(* IEC 61131-3 sources: NachHouse_CORE/V200/APP (part 8) *)

(*
   If yes = false THEN
      yTx2 := '';
      _Nh1RowTxt();
   END_IF;
*)

END_FUNCTION
(*
FUNCTION _Nh_IO4 {HIDDEN} :BOOL
	// ACT,ALA,BLK - vykona sa pred SCN. SCN mozu vstupovat do ACT....
//   _Nh_IO_INI( vz:=4);
	FOR nd := 1 TO aVaz[cf].Rec DO
		IF _NhxVaz(cv:=4, nd:=nd) THEN
//			_Nh_IO_OK();

			ok := true;
  			IF _NhxPt(c:=xVaz^.in.c,n:=xVaz^.in.n,x:=22) THEN
			  	xDev  := xPt;
			ELSE
				ok := false;
			END_IF;
	      IF _NhxPt(c:=xVaz^.ou.c,n:=xVaz^.ou.n,x:=23) THEN
				xDev2 := xPt;
			ELSE
				ok := false;
			END_IF;
			IF ok THEN
		      xDev^.al.lst   := true;                                             				// SCN ma list
   	   	xDev2^.al.lst  := true;                                             				// DEV do scn ma list
      		IF xDev^.al.ou.cmd > 0 THEN
   	   	   xDev2^.al.IN.cmd  := xDev^.al.ou.cmd;
		         xDev2^.al.IN.par  := xVaz^.ou.p;                               				// do DEV sa posle vzdy parameter ou.p
//	         xDev2^.al.IN.par  := 8;                               				// do DEV sa posle vzdy parameter ou.p

   	   	   xDev2^.al.IN.val  := xDev^.al.ou.val;                       					// parameter DEV z vazby
      		   xDev2^.al.wsb  	:= xDev^.al.wsb;                       						// zaisi pripadne blokovanie PIR pte DEV v liste
					xDev^.al.wsb		:= false;																// po prebrati vynuluje priznak WSB
		      END_IF;
			END_IF;
		END_IF;
   END_FOR;
END_FUNCTION
*)

FUNCTION _Nh_IO4  {HIDDEN}  :BOOL
	// ACT,ALA,BLK - vykona sa pred SCN. SCN mozu vstupovat do ACT....
   _Nh_IO_INI( vz:=4);
	FOR nd := 1 TO aVaz[cf].Rec DO
		IF _Nh_IO_OK() THEN
	      xDev^.al.lst   := true;                                             				// SCN ma list
      	xDev2^.al.lst  := true;                                             				// DEV do scn ma list
      	IF xDev^.al.ou.cmd > 0 THEN
   	      xDev2^.al.IN.cmd  := xDev^.al.ou.cmd;
	         xDev2^.al.IN.par  := xVaz^.ou.p;                               				// do DEV sa posle vzdy parameter ou.p
      	   xDev2^.al.IN.val  := xDev^.al.ou.val;                       					// parameter DEV z vazby
      	   xDev2^.al.wsb  	:= xDev^.al.wsb;                       						// zaisi pripadne blokovanie PIR pte DEV v liste
				// toto sa urovni az akcii v dalsom cykle
//				xDev^.al.wsb		:= false;																// po prebrati vynuluje priznak WSB
	      END_IF;
		END_IF;
   END_FOR;
END_FUNCTION

// z akcii uz vypinaju aj scenu ak je lvl=0.0 alebo ak < 100, tak zapnu len tie DEV pomerom, ktore maju v par, lvl > 0.0
FUNCTION _Nh_IO3    :BOOL
	// SCN - po ACT,(IO4) ktore mozu nastavit SCN nejaky stav
   _Nh_IO_INI( vz:=3);
	FOR nd := 1 TO aVaz[cf].Rec DO
		IF _Nh_IO_OK() THEN
	      xDev^.al.lst   := true;                                             					// SCN ma list
      	xDev2^.al.lst  := true;                                             					// DEV do scn ma list
			xScn				:= xDev;
      	IF xDev^.al.ou.cmd > 0 THEN
				IF xDev^.cf.typ = 1 THEN
      		   xDev2^.al.up  		:= xDev^.al.up;                       						// parameter DEV z vazby
					xDev2^.al.IN.cmd  := xDev^.al.ou.cmd;
		         xDev2^.al.IN.par  := xVaz^.ou.p;                               					// do DEV sa posle vzdy parameter ou.p
				ELSE
		         xDev2^.al.IN.par  := xVaz^.ou.p;                               					// do DEV sa posle vzdy parameter ou.p
   	   	   xDev2^.al.IN.val  := xDev^.al.ou.val;                       						// parameter DEV z vazby
					xDev2^.al.IN.cmd  := xDev^.al.ou.cmd;
(*
				IF xDev^.al.ou.val = 0.0 THEN
	   	      xDev2^.al.IN.cmd  := 10;
				ELSIF xDev^.al.ou.val < 100.0 THEN
	   	      xDev2^.al.IN.cmd  := 9;
					xDev^.al.Qx 		:= false;
				ELSE
	   	      xDev2^.al.IN.cmd  := xDev^.al.ou.cmd;
				END_IF;
      	   xDev2^.al.wsb  	:= xDev^.al.Wsb;                       						// parameter DEV z vazby
*)

					IF xDev^.al.ou.cmd = 11 THEN
						IF aCfg[xVaz^.ou.c].par > 0 THEN															// DEV v scene ma parameter
							IF _NhxPar(cp := aCfg[xVaz^.ou.c].par, np := xVaz^.ou.p,x:=252) = false  THEN																	   // NEnasiel sa parameter
							;
							ELSIF xPar^.all.lvl = 0 THEN						// LVL>0 ale ine ako ma byt
	   	      			xDev2^.al.IN.cmd  := 10;
							END_IF;
						END_IF;
					END_IF;
      		   xDev2^.al.wsb  	:= xDev^.al.Wsb;                       						// parameter DEV z vazby
				END_IF;
			ELSIF xDev^.cf.typ = 1 THEN																	// len rolety
				IF xDev2^.al.sta > 2  THEN
					xScn^.cx.all.LastScnOn := true;
				END_IF;
			ELSIF xDev2^.al.ou.val > 0. THEN
				xScn^.cx.all.LastScnOn := true;
(*
			ELSIF xDev^.al.Qx = false THEN																// DEV v scene je zapnute
				;
			ELSIF aCfg[xVaz^.ou.c].par > 0 THEN															// DEV v scene ma parameter
				IF _NhxPar(cp := aCfg[xVaz^.ou.c].par, np := xVaz^.ou.p,x:=252) = false  THEN																	   // NEnasiel sa parameter
					;
				ELSIF xPar^.all.lvl <> REAL_TO_USINT(xDev2^.al.ou.val) THEN						// LVL>0 ale ine ako ma byt
					// vypne scenu
//					xDev^.al.In.val 	:= 0.0;	//xDev2^.al.ou.val;
//					xDev^.al.Ou.val 	:= 0.0;	//xDev2^.al.ou.val;
					xDev^.al.Qx 		:= false;
					xDev^.al.in.cmd	:= 3;																	// vypne priznak zapnutia a resetne casy
				END_IF;
*)
			END_IF;
		END_IF;
   END_FOR;
END_FUNCTION

(*
// z akcii uz vypinaju aj scenu ak je lvl=0.0 alebo ak < 100, tak zapnu len tie DEV pomerom, ktore maju v par, lvl > 0.0
FUNCTION _Nh_IO3    :BOOL
	// SCN - po ACT,(IO4) ktore mozu nastavit SCN nejaky stav
   _Nh_IO_INI( vz:=3);
	FOR nd := 1 TO aVaz[cf].Rec DO
		IF _Nh_IO_OK() THEN
	      xDev^.al.lst   := true;                                             					// SCN ma list
      	xDev2^.al.lst  := true;                                             					// DEV do scn ma list
			xScn				:= xDev;
      	IF xDev^.al.ou.cmd > 0 THEN
				IF aCfg[xVaz^.ou.c].par > 0 THEN															// DEV v scene ma parameter
					IF _NhxPar(cp := aCfg[xVaz^.ou.c].par, np := xVaz^.ou.p,x:=252) THEN
						xScn^.me.delayOff := MAX(xScn^.me.delayOff, _Nh_N12(aCfg[xVaz^.ou.c].tgrp=31,xPar^.all.tDelay,xPar^.all.tDelay/10)+2 );	// MAX opozdene spustenie z niektoreho DEV
					ELSE
						yTx2	:= CONCAT('_Nh_IO3: Not Find par: cf:',USINT_TO_STRING(xVaz^.ou.c),',cp:',USINT_TO_STRING(aCfg[xVaz^.ou.c].par),
											', np: ',INT_TO_STRING(xVaz^.ou.p),', vz3:',INT_TO_STRING(nd)  )  ;
    					rb		:= _Nh1RowTxt(logRst := 1);
						ok1 	:= false;
					END_IF;
				ELSE	ok1 := false;
				END_IF;
 				xDev2^.al.wsb  	:= xDev^.al.Wsb;                       						// priznak WSB
				xDev2^.al.IN.cmd  := xDev^.al.ou.cmd;
  	   	   xDev2^.al.IN.val  := xDev^.al.ou.val;                       					// parameter DEV z vazby
	         xDev2^.al.IN.par  := xVaz^.ou.p;
				IF xDev^.cf.typ = 1 THEN
      		   xDev2^.al.up  		:= xDev^.al.up;                      						// pre ROL DOLEZITE !!! - nastavi smer pohybu rolety
				END_IF;
				IF xDev^.al.ou.cmd = 11 THEN
					IF ok1 = false THEN
						;
					ELSIF xPar^.all.lvl = 0 THEN						// LVL>0 ale ine ako ma byt
 						xDev2^.al.IN.cmd  := 10;
					END_IF;
				END_IF;
			ELSIF xDev^.al.ou.val = 0. THEN																// scn je vypnuta
				;
			ELSIF xDev^.cf.typ = 1 THEN																	// len rolety
				IF xDev2^.al.sta > 2  THEN
					xScn^.cx.all.LastLvl	:= 100;
				END_IF;
			ELSIF xDev2^.al.ou.val > 0. THEN
				xScn^.cx.all.LastLvl	:= 100;
			END_IF;
		END_IF;
   END_FOR;
END_FUNCTION
*)

(*

// pred Rosochom - z akcii nevypinali scenu, ked bola 0.0

FUNCTION _Nh_IO3  :BOOL
	// SCN - po ACT,(IO4) ktore mozu nastavit SCN nejaky stav
   _Nh_IO_INI( vz:=3);
	FOR nd := 1 TO aVaz[cf].Rec DO
		IF _Nh_IO_OK() THEN
	      xDev^.al.lst   := true;                                             					// SCN ma list
      	xDev2^.al.lst  := true;                                             					// DEV do scn ma list
			xScn				:= xDev;
      	IF xDev^.al.ou.cmd > 0 THEN
	         xDev2^.al.IN.par  := xVaz^.ou.p;                               					// do DEV sa posle vzdy parameter ou.p
      	   xDev2^.al.IN.val  := xDev^.al.ou.val;                       						// parameter DEV z vazby
   	      xDev2^.al.IN.cmd  := xDev^.al.ou.cmd;
      	   xDev2^.al.wsb  	:= xDev^.al.Wsb;                       						// parameter DEV z vazby
			ELSIF xDev^.al.Qx = false THEN																// DEV v scene je zapnute
				;
			ELSIF aCfg[xVaz^.ou.c].par > 0 THEN															// DEV v scene ma parameter
				IF _NhxPar(cp := aCfg[xVaz^.ou.c].par, np := xVaz^.ou.p,x:=252) = false  THEN																	   // NEnasiel sa parameter
					;
				ELSIF xPar^.all.lvl <> REAL_TO_USINT(xDev2^.al.ou.val) THEN						// LVL>0 ale ine ako ma byt
					// vypne scenu
//					xDev^.al.In.val 	:= 0.0;	//xDev2^.al.ou.val;
//					xDev^.al.Ou.val 	:= 0.0;	//xDev2^.al.ou.val;
					xDev^.al.Qx 		:= false;
					xDev^.al.in.cmd	:= 3;																	// vypne priznak zapnutia a resetne casy
				END_IF;
			END_IF;
		END_IF;
   END_FOR;
END_FUNCTION
*)

(*
FUNCTION _Nh_IO3  :BOOL
	// SCN - po ACT,(IO4) ktore mozu nastavit SCN nejaky stav
   _Nh_IO_INI( vz:=3);
	FOR nd := 1 TO aVaz[cf].Rec DO
		IF _Nh_IO_OK() THEN
	      xDev^.al.lst   := true;                                             					// SCN ma list
      	xDev2^.al.lst  := true;                                             					// DEV do scn ma list
      	IF xDev^.al.ou.cmd > 0 THEN
   	      xDev2^.al.IN.cmd  := xDev^.al.ou.cmd;
	         xDev2^.al.IN.par  := xVaz^.ou.p;                               					// do DEV sa posle vzdy parameter ou.p
      	   xDev2^.al.IN.val  := xDev^.al.ou.val;                       						// parameter DEV z vazby
//      	   xDev2^.al.wsb  	:= xDev^.cx.all.LastWsb;                       						// parameter DEV z vazby
      	   xDev2^.al.wsb  	:= xDev^.al.Wsb;                       						// parameter DEV z vazby

//  	   	ELSIF xDev^.al.Qx THEN 												      						// test SCN ci je ON/OFF, povoli sa ked je scena v pokoji Qx=true
  	   	ELSIF xDev^.cx.all.LastScnOn THEN 												      						// test SCN ci je ON/OFF, povoli sa ked je scena v pokoji Qx=true
				// ak aspon jedno DEV nema hodotu aku ma mat v scene = vypne scenu
				IF xDev^.al.ou.val > 0.0  THEN																// scena je zapnuta
					IF aCfg[xVaz^.ou.c].par > 0 THEN															// DEV v scene ma parameter
    					IF _NhxPar(cp := aCfg[xVaz^.ou.c].par, np := xVaz^.ou.p,x:=252) = false THEN
							;
						ELSIF xPar^.all.lvl <> REAL_TO_USINT(xDev2^.al.ou.val) THEN						// kazde DEV v SCN-liste musi mat aktualny LVL = parametru

							xDev^.cx.all.LastScnOn	:= false;														// ak sa najde prva nezhoda, tato SCN sa oznaci a OFF
							xDev^.al.sta 				:= 0;                                              // a uz sa s nou tu nepracuje
							xDev^.al.IN.val 			:= 0.0;															// vypne scenu
							xDev^.al.OU.val 			:= 0.0;
      					/////15.9.24	vypne prebiehajuce casy vypnutia
//							xDev^.al.et 	:= 0;																	// cas od PIR
//							xDev^.al.ex 	:= 0;																	// max.cas zapnutia
						END_IF;
					END_IF;
				END_IF;
			END_IF;
		END_IF;
   END_FOR;
END_FUNCTION
*)

FUNCTION _Nh_SVX_CMD_1     : BOOL
	IF xDev^.al.in.CMD = 3 THEN         										// len nastavilo proznak vypnutia a resetlo casy
		;
	ELSIF xDev^.al.in.CMD > 0 THEN         										// povolene prikazy testuju blokovanie PIR a oneskorenie
			xDev^.al.Off 			:= xDev^.al.OU.val = 0.0 AND xDev^.al.IN.val > 0.0; // je vypnute a ma sa zapnut - pre lampu, ktora ma dlhy nabeh z OFF->ON
			xDev^.cx.all.LastWsb	:= xDev^.al.wsb;										// prisiel z wsb
			IF xDev^.al.RUN = 255 THEN   													// Koniec Delay
				xDev^.al.RUN := 0;
 			ELSIF xPar^.all.tDelay > 0 THEN 												// opozdene vykonanie
	   	   xDev^.al.RUN   	:= xDev^.al.in.CMD;                              			// po skonceni opozdenia sa zoberie LVL z parametri - tu pridu len DEV s parametrom
				xDev^.al.in.CMD	:= 0;
   	   	xDev^.al.et    	:= xPar^.all.tDelay ;                        //
  	   		xDev^.al.CM    	:= 2;                                        // vykonava sa opozdenie
   	   	xDev^.al.ct    	:= 3;                                     	// Delay je vzdy v [100ms]
   		END_IF;
		   IF xDev^.al.in.CMD = 1 THEN                                    	// prepnut WEB/WSB
         	xDev^.al.in.val   := vr;
      		IF xDev^.al.ou.val > 0.0 THEN                               	// je zapnute, treba vypnut z WEB/WSB
         		xDev^.al.in.val   := 0.0;
				ELSIF xPar^.all.lvl = 0 THEN
           		xDev^.al.in.val	:= 100.0;                              // zapnut naplno
					xPar^.all.lvl 		:= REAL_TO_USINT(xDev^.al.in.val);				// nastavi LVL v prametri - najma pri vazbach
      		ELSE
					xDev^.al.in.val := USINT_TO_REAL(xPar^.all.lvl);				// nastavi LVL v prametri - najma pri vazbach
      		END_IF;
      		_Nh_Dev_RMP();
   		END_IF;
		   IF xDev^.al.in.CMD > 0 THEN         										// povolene prikazy testuju blokovanie PIR a oneskorenie
			   _NhxRom(nr := xDev^.cf.rom, x:=-10);
			   IF xDev^.al.wsb = false THEN                                   // nic sa nedeje neprislo z WSB {mozno z ACT..SCN}
   			   ;
	   		ELSIF  xDev^.al.in.val > 0.0 AND xPar^.all.BlPirON THEN       	// je ON
   	   		xRom^.me.BlPirOn    := 50;  	                             	// zapnutie od WSB/WEB vzdy blokuje PIR
   	   		xRom^.me.BlPirOff   := 0;                               		// resetne sa cas blokovania po vypnuti
	   		ELSIF xPar^.all.BlPirOff AND xRom^.cx.BlPirOFF > 0 THEN 			// kontrola na blokovanie PIR po vypnuti WSB/WEB
   				xRom^.me.BlPirOff := MAX(xRom^.me.BlPirOff,xRom^.cx.BlPirOFF); // max cas blokovania po vypnuti
	   		END_IF;
				// casy vypnutia
	         IF xDev^.al.IN.val < 1.0 THEN                   		// ma sa vypnut
					xDev^.al.IN.val 	:= 0.0;
   	      ELSIF xDev^.al.OU.val < 1.0 THEN                      // je OFF a ma za zapnut
      	      xDev^.al.ex := UINT_TO_INT(xDev^.cx.all.tMaxON);   // max cas zapnutia [min] - pohyb neresetuje
         	END_IF;
	         IF xDev^.al.IN.val > 0.0 THEN
					xDev^.al.up		:= true;
      	      IF xPar^.all.tOff > 0 THEN
         	      xDev^.al.et := xPar^.all.tOff;                  // vypnut po cas
            	   xDev^.al.ct := 3;                               // po 100mSEC
	            ELSE
   	            xDev^.al.et := 0;                               // nema sa vypnut po case
      	      END_IF;
				ELSE
					xDev^.al.ex    	:= 0;
				 	xDev^.al.et    	:= 0;
				END_IF;
				_Nh_Dev_CMD();			                                 // vyvolat zapnutie HW cez CMD
			END_IF;
	END_IF;

END_FUNCTION

FUNCTION _Nh_SVX_Qx    : BOOL
	_Nh_SVX_Qx := false;
	IF _Dev_Qx_PAR(dpa:=xDev^.cf.par) THEN

		_Nh_SVX_Qx := true;
		xDev^.al.el		:=	0;
		xDev^.al.CM    := 0;													// ak bezi delay cm:=2, novy prikaz ho zrusi
//		xDev^.al.RUN   := 0;	                                    //

		IF aCfg[cf].par > 0 THEN											// dev ma parameter, SIR napr nema parameter
 	   	vr    := USINT_TO_REAL(xPar^.all.Lvl);                // default sa podhodi LVL
		ELSE
			vr := 0.0;                                          	// bez parametra nebude potrebovat, lebo pride konkretne CMD
		END_IF;

		xDev^.cx.all.LastCMD 	:= xDev^.al.in.CMD;					// zapamata posledny pokyn
// 		xDev^.cx.all.LastCMDin	:= true;                         // pokyn je prichadzajuci

		CASE xDev^.al.in.CMD OF
	      1: // prepnut z WEB
   	      xDev^.al.wsb      := true;									// nasilne sa podhodi ako z WSB, aby sa zablokoval pir
//      	   xDev^.al.in.CMD   := 1;
	      2: // prepnut z WSB												// wsb nastavi priznak WSB vo vazbach automaticky
   	      xDev^.al.in.CMD   := 1;
      	3: // resetovat casy nastavit OFF, ale neposielat nic
				cmd	:= 0;
				_Nh_Dev_OFF(cmd:=3);
				xDev^.al.in.CMD := 0;

			6: // stmievanie z  WSB - start
   	      IF xDev^.al.ou.VAL > 0.0 THEN								// stmieva sa len, ak je ON
      	      xDev^.al.Up    := NOT xDev^.al.Up;
					IF xDev^.al.ou.VAL <= 1.0 THEN
      	      	xDev^.al.Up    := true;
					ELSIF xDev^.al.ou.VAL > 99.0 THEN
    					xDev^.al.Up    := false;
					END_IF;
					IF aCfg[cf].lvl254 THEN
	         	   xDev^.al.rmp   := 1;                            // doladit ???
					ELSE
	         	   xDev^.al.rmp   := 3;
   				END_IF;
	  			ELSIF _NhxRom(nr := xDev^.cf.rom, x:=-13) THEN					// ak svetlo nesvieti, PRESS zrusi blokovanie
      	      xRom^.me.BlPirOn 	:= 0;
         	   xRom^.me.BlPirOff := 0;
					xDev^.al.cm := 255;								// aby sa uz az do pustenia BTN nic nerobilo
	         END_IF;
				xDev^.cx.all.LastLvl	:= REAL_TO_USINT(xDev^.al.Ou.val);
				xDev^.al.in.CMD		:= 0;

   	   7: // slider SVA
				IF aCfg[cf].lvl254 THEN
         	   xDev^.al.rmp   := 1;                            // doladit ???
				ELSE
         	   xDev^.al.rmp   := 2;
  				END_IF;
				xDev^.cx.all.LastLvl	:= REAL_TO_USINT(xDev^.al.Ou.val);
				xDev^.al.in.CMD		:= 0;
				xDev^.al.CM				:= 7;

	      8: // RGB - vyber farby a slidery RGBWA
   	      xDev^.al.rmp      := 0;
				xDev^.al.in.CMD	:= 0;

	      9: // specialne zapnutie/vypnutie
				// ak  je prichadzajuci LVL = 0, tak vypne,
				// ak lvl < 100 tak zapne na pomer k hodnoty z parametra
				// ak lvl = 100% tak zapne na plny parameter
				IF vr  = 0.0 THEN
					xDev^.al.in.val := 0.0;
				ELSIF xDev^.al.in.val < 100.0 THEN
					xDev^.al.in.val := vr * xDev^.al.in.val * 0.01;
				ELSE
					xDev^.al.in.val := vr;
				END_IF;
				_Nh_Dev_RMP();

	     10: // OFF + zapnut blokovanie PIR
   	      xDev^.al.in.val   := 0.0;

	     11: // zapnutie na 100%
				xDev^.al.in.val   := 100.0;                              // zapnut naplno
				_Nh_Dev_RMP();

	     12: // blikac - priame zapnutie na LVL z parametra ak al.in.val > 0, iba vypnut , bez kontroly casov
   	     	xDev^.al.IN.val   := vr;
      	   xDev^.al.wsb      := false;								// nasilne sa podhodi ako z WSB, aby sa zablokoval pir
				_Nh_Dev_RMP();

	     13: // zapnutie na to co je al.in.val (blikac), bez kontroly casov
				_Nh_Dev_RMP();

		  14: // zapnut na LVL, ulozenu v parametri, nastavit casy opozdeny start/po case vypnut/max.cas zapnutia
   	      xDev^.al.in.val   	:= vr;
				_Nh_Dev_RMP();

	     15: // len zapamatat/ulozit aktualnu LVL pre dalsiu obnovu (blikac)
				xDev^.cx.all.LastLvl := REAL_TO_USINT(xDev^.al.OU.Val);
				xDev^.al.in.CMD	:= 0;
				xDev^.al.trg.Q  	:= 0;													// aby CMD v dalom cykle vyhodnotilo ako Qr, nieQ
				xDev^.al.trg.Qf 	:= 0;

   	  16: // obnovit zapamatany LVL po ukonceni blikaca
				xDev^.al.In.Val		:= USINT_TO_REAL(xDev^.cx.all.LastLvl);
				_Nh_Dev_CMD();			                                 // vyvolat zapnutie HW cez CMD
				xDev^.al.in.CMD	:= 0;

	     21: // PIR - ON
   	      _NhxRom(nr := xDev^.cf.rom, x:=-14);
      	   IF xRom^.me.BlPirOn = 0 AND xRom^.me.BlPirOFF = 0 THEN  	// nie je blokovana ROM po vypnuti, ani po zapnuti
         	   IF xDev^.al.ou.Val < 0.9 OR xPar^.all.rPir THEN          	// je OFF alebo bezi cas-to-OFF a pohyb resetuje cas
            	   xDev^.al.IN.val   := vr;
						_Nh_Dev_RMP();
						xDev^.al.CM				:= 14;
   	         END_IF;
      	   ELSE
	      	   xDev^.al.in.CMD   := 0;
   	      END_IF;
      	   xDev^.al.wsb      := 0;

			{$IFDEF __NH_DALI}

   	   43: // ON/OFF DLS + dali 5 in On
				xDLs	:= xDev;
	         IF xDls^.cx.cfg.out5inOne THEN 										// 5 in On
					IF xDev^.al.OU.val > 0.0 THEN										// je zapnute, treba vypnut
						ii						:= 0;
					ELSE
						ii						:= 254;
					END_IF;
					FOR i := 1 TO 5 DO
						xPar^.rgb.lvl[i] := ii;          							// default parameter je namapovany
   	  			END_FOR;
					xDev^.al.in.val 	:= 100;                                // vzdy posle prikaz do DLM
	      	   xDev^.al.rmp      := 0;
					cmd					:= 143;
					xDev^.al.in.CMD	:= 0;
   	      ELSE

      	   END_IF;

	     143: // DLS 5-In-One pokyn z {TVE} nastavenych na RGBWA
				xPtIO 	:= UDINT_TO_PTR( REAL_TO_UDINT(xDev^.al.in.val) ) ;	   		// prenasa sa adresa IO, pre zistenie farby
				IF xPtIO^.val > 0. THEN																	// zapnut
					ii	:= 254;
				ELSE
					ii	:= 0;
				END_IF;
				IF xPtIO^.dev.o > 0 THEN                                                // zisti sa, ktora farba sa nastavika
//						xPar^.rgb.lvl[xPtIO^.dev.o] := MIN(254,REAL_TO_USINT(xPtIO^.val));   // nastavi sa LVL, vzdy 254
					xPar^.rgb.lvl[xPtIO^.dev.o] := ii;   											// nastavi sa LVL, konkretnehj farby RGBWA vzdy 254
				END_IF;
//				xDev^.al.in.val	:= 255.0;                                               // vzdy vysle sa prikaz - aktualizuje vsetky farby
				xDev^.al.in.val 	:= 100;                                // vzdy posle prikaz do DLM
				cmd					:= 143;
				xDev^.al.in.CMD	:= 0;

	     144: // DLS 5-In-One dotyk nad konkretnou farbou znamen vyslat to co tam je
//				xDev^.al.in.val 	:= 255.0;
				xDev^.al.in.val 	:= 100;                                // vzdy posle prikaz do DLM
				xDev^.al.in.CMD	:= 0;
   	   	cmd       			:= 143;
			{$END_IF}
   	ELSE
			;
   	END_CASE;
//		_Nh_SVX_CMD_1();

	ELSIF xDev^.al.trg.Q THEN                                         // presss alebo len zopar cyklov, ked sa neuvolni cmd

		IF aCfg[cf].lvl254 THEN	                                       // DALI
			ok	 	:= (SYSTEM_S.R_EDGE_500MS OR SYSTEM_S.F_EDGE_500MS);  // vysiela sa kazdy 250ms
			kr 	:= 7.;
//			kr 	:= 1.;
			ur		:= 100.;
		ELSE
			ok	 	:= aSys.PULSE_50MS;	//SYSTEM_S.R_EDGE_100MS;			// kazdych 50ms, alebo podla cyklu
			kr 	:= 1.;
			ur		:= 100.;
		END_IF;

		IF xDev^.al.up = false THEN
			kr	:= kr * -1.;
		END_IF;
		cmd	:= 0;
		IF xDev^.al.cm = 255 THEN                                      // press, ked svetlo nesvietilo {zrusenie blokovania}
			;
		ELSIF ok = false THEN														// nenastala casova vzorka
			;
		ELSIF xDev^.cx.all.LastCMD = 6 THEN										// drzi sa WSB
			vr						:= xDev^.al.IN.val + kr ;
  			IF vr > 100. THEN
				vr := 100.;
			ELSIF vr < 1. THEN
				vr := 1.;
			END_IF;
			xDev^.al.IN.val	:= LIMIT(1.0, vr, ur);
			IF vr <> xDev^.al.IN.val THEN                              	// uz sa dosiahol niektory limit
				xDev^.al.cm := 255;
			ELSE
				_Nh_Dev_CMD();
			END_IF;
		ELSIF xDev^.cx.all.LastCMD = 7 THEN	                           // slider
			IF ABS(xDev^.al.ou.val - xDev^.al.In.val) >= ABS(kr)  THEN  // bude vysielat do HW, len ked je zmena vacsia
	 			_Nh_Dev_CMD();
			END_IF;
		ELSIF xDev^.cx.all.LastCMD = 8 THEN	                           // RGB
 			_Nh_Dev_CMD();
		END_IF;

	ELSIF xDev^.al.trg.Qf THEN														// koniec CMD
		xDev^.al.wsb 	:= 0;
		IF xDev^.cx.all.LastCMD = 8 	OR									// zmena fazby = vyber predvolby
			xDev^.al.cm = 255				OR                         // prikaz uz bol vykonany
			(xDev^.cx.all.LastCMD >= 4 AND xDev^.cx.all.LastCMD <= 7) THEN	// 4=SW-Dim,6=WSB-dim,7-slider
			xDev^.al.cm		:= 0;
			xDev^.al.et		:= 0;

//			_NhxPar(cp := aCfg[cf].par , np := xDev^.al.ou.par, cf:=cf, nd:=nd, x:=110);

			xPar^.all.lvl := REAL_TO_USINT(xDev^.al.in.val);		// zapamata LVL v default parametri
			_Nh_Dev_CMD();														// este raz posle, lebo slider nemusel zachytit vsetko
		END_IF;

	ELSIF aSys.Restart THEN
		IF xDev^.cf.LvlOnRst  THEN	 								// po restarte obnovit
			_Nh_Dev_CMD();			                                 // zapnut HW
		ELSE
//			xDev^.al.in.Val := 0.0;                               // vypnut aj IN
		END_IF;
	END_IF;
END_FUNCTION

FUNCTION _Nh_SVX   : BOOL
	VAR_INPUT
		c		: 	USINT;
	END_VAR
	VAR_TEMP
		i		: USINT;
//		ii		: USINT;
	END_VAR
   _Nh_SVX	:= _Dev_INI(c := c);
	nd			:= 1;
   WHILE nd <= aCfg[cf].Rec DO
      IF _Nh_Dev_REC(blk:=true) THEN //AND nd = 2 THEN
			IF _Nh_SVX_Qx() THEN
				_Nh_SVX_CMD_1();																// nie pre SCN
			END_IF;
		   xDev^.al.IN.CMD   := 0;															// reset vstup, aby s v dalsom kole vyhodnotil Q,Qf
			IF xDev^.al.cm = 2 THEN
				cmd	:= 0;
				IF _Nh_Dev_ET_UINT(t :=3, et:= ADR(xDev^.al.et) ) THEN			// odpocitava Delay [min]
					xDev^.al.in.cmd	:= xDev^.cx.all.LastCMD;
					xDev^.al.in.par	:= xDev^.al.ou.par;
					xDev^.al.RUN		:= 255;
//					xDev^.al.cm 		:= 0;
				END_IF;
			ELSIF xDev^.al.cm = 255 THEN													// bezi press a uz sa nema co vykonat
				cmd	:= 0;
			ELSIF _Nh_Dev_ET_UINT(t :=3, et:= ADR(xDev^.al.et) ) OR				// odpocitava cas zapnutia [min]
 					_Nh_Dev_ET_INT (t :=2, et:= ADR(xDev^.al.ex) ) THEN			// odpocitava max cas zapnutia [min]
				_Nh_Dev_OFF(cmd:=0);
				_Nh_Dev_CMD();			                                 			// zapnut HW
			END_IF;
//			ok3	:= true;
			ok3	:= cf <> 42;																// stav DALI-mastra sa robi inak ako cez _Nh_Sta_Rom
			CASE cmd OF
           	 0: ;
				 3: ; //
          	10: ; // SVD,ZAS,SIR.... digital
			      	xSvD 					:= xDev;
						IF xSvD^.hw.d[0] > 0 THEN
	                  xDev^.al.Ou.CMD	:= 180;
   	   			   xPtB 					:= UDINT_TO_PTR(xSvD^.hw.d[0]);

 							_Nh_Log_Evn_ADD(tsk:=10);

      				   xDev^.al.OU.val   := xDev^.al.IN.val;
         			 	xPtB^             := REAL_TO_BOOL(xDev^.al.OU.val);                  // in, nie ou
	 	      		   IF xDev^.cf.inv THEN
 		         			xPtB^ := NOT xPtB^;
	      	  	   	END_IF;
						END_IF;

				11:	// SVA
    					xDev^.al.Ou.CMD	:= 180; 																	// default CMD pre vystupne zariadenie
						IF xDev^.hw.typ = 43 THEN
							;
						ELSIF xDev^.hw.d[0] > 0  THEN                                     			// xDev = xSva
							ok := xDev^.cx.dim.DimHW;
							IF ok THEN                                                        // ma sa stmievat HW
								IF xDev^.hw.d[1] = 0 THEN                                     	// ak nie je HW adresa stmievania
									ok := false;                                                // bude sa stmievat SW
								END_IF;
							ELSIF xDev^.hw.d[1] > 0 THEN                                     	// ma sa stmievat SW ale mame HW adresu rampy
								xPtU 					:= UDINT_TO_PTR(xDev^.hw.d[1]);
								xPtU^ 				:= 0;														// rampu nastavi na 0
							END_IF;

 							_Nh_Log_Evn_ADD(tsk:=10);

							IF ok THEN
								xPtU 					:= UDINT_TO_PTR(xDev^.hw.d[1]);
								xPtU^ 				:= xDev^.al.rmp;
   	   		         xDev^.al.ou.val   := xDev^.al.in.val;
							ELSE
								_Nh_Dim_SW();
							END_IF;
							xDev^.al.el			:= 0;
							xPtR 					:= UDINT_TO_PTR(xDev^.hw.d[0]);
							xDev^.al.ou.val	:= LIMIT(0.0, xDev^.al.in.val, 100.0);
							xPtR^					:= _Nh_LVL_100(	lvlMin	:=	xDev^.cx.sva.Lv0,
																			lvlMax	:=	xDev^.cx.sva.Lv1,
																			lvlIn		:=	xDev^.al.ou.val);
							CASE xDev^.hw.typ OF
      	              0:	// BOOL
									xPtB	:= xPtr;
									xPtB^	:= REAL_TO_BOOL(xPtr^);
                    	  1: // REAL
//							  		xPtR^	:= kr;
							  2:	// USINT
									xPtU	:= xPtr;
									xPtU^	:= REAL_TO_USINT(xPtr^);
      	            END_CASE;
						END_IF;

(*

                  xDev^.al.Ou.CMD	:= 180; 																	// default CMD pre vystupne zariadenie
						IF xDev^.hw.d[2] > 0 THEN                                     		// mame adresu HW minima (RLC)
 							xPtR 	:= UDINT_TO_PTR(xDev^.hw.d[2]);
							xPtR^ := _Nh_255_100(xDev^.cx.sva.Lv0);
						END_IF;
						xPtR := UDINT_TO_PTR(xDev^.hw.d[0]);
						IF xDev^.cx.dim.DimHW THEN														// stmieva sa HW - treba mat na to HW !!!!
							IF xDev^.hw.d[1] = 0 THEN                                     	// ak nie je HW adresa
								xDev^.cx.dim.DimHW := 0;
							ELSE
		    					xPtU := UDINT_TO_PTR(xDev^.hw.d[1]);
							END_IF;
						END_IF;
					   IF xDev^.al.off AND xDev^.cx.dim.tOnL > 0	THEN	     					// prve zapnutie lampy, ktora ma opozdeny nabeh
							xDev^.al.run		:= xDev^.al.cm;
							xDev^.al.cm			:= 2;                                        // delay
							xDev^.al.et		   := USINT_TO_UINT(xDev^.cx.dim.tOnL);
							xDev^.al.ct		   := 3;
							xDev^.al.ou.val   := USINT_TO_REAL(xDev^.cx.sva.Lv0);				// mSec
							IF xDev^.cx.dim.DimHW THEN
			               xPtU^ 				:= 0;													// bez rampy
							END_IF;
						ELSIF xDev^.cx.dim.DimHW THEN
		               xPtU^ 				:= xDev^.al.rmp;
      	         	xDev^.al.ou.val   := xDev^.al.in.val;
						ELSIF xDev^.al.cm = 4 THEN
							xDev^.al.cm := xDev^.al.RUN;
						ELSE
							xDev^.al.up := xDev^.al.in.val > xDev^.al.OU.val;
							xDev^.al.cm := 4;
						END_IF;
						xDev^.al.ou.val			:= LIMIT(0.0, xDev^.al.ou.val, 100.0);
*)

				12:  // RGB

            	   xDev^.al.Ou.CMD	:= 180;
						xRgb					:= xDev;
						xDev^.al.ou.val	:= LIMIT(0.0, xDev^.al.in.val, 100.0);
   		      	vr	:= _Nh_LVL_100(	lvlMin	:=	xDev^.cx.sva.Lv0,
													lvlMax	:=	xDev^.cx.sva.Lv1,
													lvlIn		:=	xDev^.al.ou.val);

							 _Nh_Log_Evn_ADD(tsk:=10);

//						_NhxPar(cp := aCfg[cf].par , np := xDev^.al.ou.par,cf:=cf, nd:=nd ,x:=-1019);       // parameter z vazby
						FOR i := 1  TO 5 DO
							IF xRgb^.hw.d[i-1] > 0 THEN
								xPtR 	:= UDINT_TO_PTR(xRgb^.hw.d[i-1]);
		   	 				xPtU 	:= xPtR;
		    					xPtU 	:= xPtU + 4;
								xPtU^ := xDev^.al.rmp;
								xPtR^ := LIMIT(0.0, (USINT_TO_REAL(xPar^.rgb.lvl[i])/255.0) * vr, 100.) ;
							END_IF;
               	END_FOR;
         254 : ; // DevExt
           ;
			ELSE
				xDev^.al.Ou.CMD	:= 0;
			END_CASE;
			///// toto je pokus 21.12.24 pri oprave stmievania cez DIM {presunute do ELSE}
			{$IFDEF __NH_DALI}
			CASE cf OF
			  	42: 	// DALI MASTER DLma
						xDLm	:= xDev;
						IF xDLm^.al.sta < 2 THEN										// NE-bezi QUERY, alebo RND
							IF cmd = 42 THEN
								dlma := INT_TO_USINT(nd);
     							_Nh_DL_ADD_Task(wht:=2, sha:=255, par:= 20, val:=xDev^.al.rmp, dlm:=dlma);				// rampa
								_Nh_DL_ADD_Task(wht:=1, sha:=255, lvl:=xDev^.al.IN.val, dlm:=dlma ); // lvl
								xDLm^.me.lvl255 	:= true;                                                          // priznak mastra
								xDLm^.me.Rmp255 	:= xDev^.al.rmp;                                                  // aka rampa do vsetkych DLS
				      	   _NhMemSetPTR(size := SIZEOF(NH_DLM_GRP), dest:= ADR(xDLm^.me.scn) );						// vynuluje sceny
							ELSE
								xDLm^.al.In.val 	:= 0.0;											// vynuluje sa, LVL urobi az sumarne DLs
							END_IF;
							xDev^.al.OU.val	:= xDev^.al.IN.val;
							xDLm^.al.sta	:= 0;                               			// stav	sa urobi az v DLs
						END_IF;
//						ok3 := 0;                               								// nevyhodnoti sta, to az kazde DEV

				44:	// DLg sa robi pred DLs ( ballastom )
    					xDLg 					:= xDev;
				  		dlma 					:= _Nh_DL_sha(nd:=nd, gr:=true, ma:=true);   // 1..2
	              	dlsl 					:= _Nh_DL_sha(nd:=nd, gr:=true);     			// 100..115
						_NhxDLm(dlm:=dlma);															// namapuje xDLm
						IF xDLm^.me.lvl255 THEN														// prikaz z mastra oznaci len v SW sceny vypnute, nic neposiela do HW
							xDev^.al.IN.val := 0.0;
						ELSIF cmd = 44 THEN
	 						IF xDLg^.me.rmp <> xDev^.al.rmp THEN                   		// zmena rampy
		         			_Nh_DL_ADD_Task(wht:=2, sha:=dlsl, par:= 20, val:=xDev^.al.rmp, dlm:=dlma);			// rampa dp vsetkych ballastov v scene
	   						xDLg^.me.rmp := xDev^.al.rmp;
   		   	      END_IF;

							IF xDev^.al.IN.val > 99.0 THEN								      // zapnut celu scenu na LVL ballastov v scene, na nizsi Level sa drobi v DLs
								_Nh_DL_ADD_Task(wht:=7, sha:=dlsl, par:=dlsl-100, dlm:=dlma );	// par je GRP 0..15,  sha je skupinova adresa 100..115
							ELSE	//IF xDev^.al.IN.val = 0. THEN											// len vypnut
								_Nh_DL_ADD_Task(wht:=1, sha:=dlsl, dlm:=dlma, lvl:=xDev^.al.IN.val );  // sha je skupinova adresa 100..115
							END_IF;

      					// v mastri oznaci, ze bol set sceny
							xDev^.al.Qx						:= true;									// priznak, ze scena je zapnuta
							xDLm^.me.scn.SET[dlsl-100] := true;									// priznak nastavene sceny
							xDLm^.me.scn.LVL[dlsl-100] := REAL_TO_USINT(xDev^.al.IN.val);
							xDLm^.me.scn.RMP[dlsl-100] := xDLg^.me.rmp;						//	ramapa do vsetkych SHA

						ELSIF xDLm^.me.scn.LVL[dlsl-100] > 0  THEN							// SCN je zapnuta
							IF xDLm^.me.scn.DEV[dlsl-100] = false THEN						// ziadne DEV v SCN NIE-je zanute aspon na minimum
								xDLm^.me.scn.LVL[dlsl-100] := 0;									// toto musi byt koli xDlG^.al.in.CMD 	:= 3;
								xDlG^.al.in.CMD 				:= 3;									// len vypne scenu a resetne casy, ALE NEPOJDE DALEJ DO PRIKAZU !!!
							END_IF;
						END_IF;
						xDLm^.me.scn.DEV[dlsl-100] := false;
						xDev^.al.OU.val	:= xDev^.al.IN.val;

				43:	// na konci urobi ballast , sumare do mastra aj skontroluje scenu
						xDLs	:= xDev;
  		            dlsl 	:= _Nh_DL_sha(nd:=nd);              								// 0..64 pre master
     					dlma 	:= _Nh_DL_sha(nd:=nd, ma:=true);          						// 1..2
						_NhxDLm(dlm := dlma);                              					// xDLm

						IF xDLm^.me.lvl255 THEN															// bol centralny LVL, ma najvyssiu prioritu
							xDev^.al.In.Val	:= xDLm^.al.Ou.Val;           					// do ballastu zapise LVL z mastra
     						xDLs^.me.rmp 		:= xDlm^.al.rmp;                             // preberie sa aj rampa, ktoru nastavil master do vsetkych SHA
							xDev^.al.OU.Val 	:= xDev^.al.IN.Val;
						ELSIF cmd = 43 THEN									      					// klasicke dev
							IF xDLs^.me.rmp <> xDev^.al.rmp THEN
 								_Nh_DL_ADD_Task(wht:=2, sha:=dlsl, par:= 20, val:=xDev^.al.rmp, dlm:=dlma);
      						xDLs^.me.rmp := xDev^.al.rmp;
           				END_IF;
							_Nh_DL_ADD_Task(wht:=1, sha:=dlsl, lvl:=xDev^.al.IN.val, dlm:=dlma );
							xDev^.al.OU.Val 	:= xDev^.al.IN.Val;
						ELSIF  cmd = 143 THEN 															// len pre xDLs^.cx.cfg.out5inOne
							xDev^.al.et 	:= 0;
							xDev^.al.ex 	:= 0;
	         			xDLs^.al.rmp   := 0;                                        // tu sa nestmieva, ide sa na ON/OFF
							IF xDLs^.me.rmp <> xDLs^.al.rmp THEN
  								_Nh_DL_ADD_Task(wht:=2, sha:=dlsl, par:= 20, val:=xDev^.al.rmp, dlm:=dlma);
       						xDLs^.me.rmp := xDev^.al.rmp;
	           			END_IF;
							xDLs^.me.SendDLM := true;
							_Nh_DL_ADD_Task(wht:=6, sha := dlsl, dlm := dlma, lvl := xDev^.al.IN.Val  );
							// zistit stav
							xDev^.al.Ou.Val := 0.0;     											// na zaciatku podhodi sa vypnute
							FOR i := 1 TO 5 DO
								IF xPar^.rgb.lvl[i] > 0 THEN          							// default parameter je namapovany
//									xDev^.al.Ou.Val := 254;											// ak je nieco z RGBWA zapnute, je cely SHA zapnuty
									xDev^.al.Ou.Val := 100.;										// ak je nieco z RGBWA zapnute, je cely SHA zapnuty
									EXIT;
								END_IF;
          				END_FOR;
							xDev^.al.In.Val := 0.0;													// u tohto typu vynuluje vstup

						// ponastavuje DLg
						ELSIF xDLs^.cx.scn.grp <> _eBtn15 THEN									// patri do nejakej sceny
                  	FOR i := 0 TO 15 DO
								IF xDLs^.cx.scn.grp[i] THEN										// patri do sceny i
									_NhxDLg(grp := i, dlm := dlma);								// namapuje scenu
									IF xDLm^.me.scn.set[i]	THEN									// scena bola v tomto cykle ON alebo OFF
										IF xDLg^.al.Ou.Val < 100. THEN                 		// scena pola stmievana, toto dev sa nezaplo/nevyplo
											xDev^.al.IN.Val := xDLg^.al.Ou.Val;					// scena nastavila len lvl, nezapla DEV
										ELSE
											xDev^.al.IN.Val := USINT_TO_REAL(xDLs^.cx.scn.lvl[i]);	// toto DLs sa nastavilo na LVL, ktoru ma urcenu v SCENE
										END_IF;
										xDLs^.me.rmp 		:= xDLm^.me.scn.RMP[i];				// scena vzdy nastavi rmpu kazdeho DLs
										xDev^.al.OU.Val 	:= xDev^.al.IN.Val;
										xDLm^.me.scn.DEV[i] := true;
//									ELSIF xDlg^.al.Qx = false THEN								// uz bola vypnuta scena predchadzajucin DEV
										;
									ELSIF xDLs^.cx.scn.lvl[i] > 0 AND xDev^.al.Ou.Val > 0. THEN // DEV ma mat uroven a je vypnute
//										xDlg^.al.Qx 		:= false;
										xDLm^.me.scn.DEV[i] := true;
//										xDlG^.al.in.CMD 	:= 3;										// len vypne scenu a resetne casy

(*
									ELSIF xDev^.al.Ou.Val = 0 AND xDLs^.cx.scn.lvl[i] > 0 THEN // DEV ma mat uroven a je vypnute
										xDlg^.al.Qx 		:= false;
										xDlG^.al.in.CMD 	:= 3;										// len vypne scenu a resetne casy
*)

(*
									ELSIF xDlg^.al.Qx = false THEN
										;
									ELSIF xDLg^.al.Ou.Val < 100. THEN                 		// scena pola stmievana, toto dev sa nezaplo/nevyplo
										IF xDev^.al.Ou.Val <> xDLg^.al.Ou.Val THEN  // dev ma iny LVL ak o ma mat v ecene
											xDlg^.al.Qx 		:= false;
											xDlG^.al.in.CMD 	:= 3;										// len vypne scenu a resetne casy
										END_IF;
									ELSIF REAL_TO_USINT(xDev^.al.Ou.Val) <> xDLs^.cx.scn.lvl[i] THEN  // dev ma iny LVL ak o ma mat v ecene
										xDlg^.al.Qx 		:= false;
										xDlG^.al.in.CMD 	:= 3;										// len vypne scenu a resetne casy
*)
									END_IF;
								END_IF;
							END_FOR;
						END_IF;

						IF xDLm^.al.sta < 2 AND xDLm^.me.lvl255 = false THEN         		// zapise priznak do mastra, ak neprebieha CHK alebo nebol centralny prikaz
							xDLm^.al.In.Val	:= MAX(xDLm^.al.In.Val, xDev^.al.IN.Val); 	// do mastra zapise hodnotu z ballastu
 			  				xDLm^.al.Ou.Val 	:= xDLm^.al.In.Val;
							IF xDLm^.al.Ou.Val > 0.0 THEN
								xDLm^.al.sta	:= 1;															// az tu sa oznaci master, ze svieti
							END_IF;
						END_IF;
			ELSE
				xDev^.al.Ou.CMD	:= 0;
			END_CASE;
			{$END_IF}

			IF ok3 THEN
				_Nh_Sta_Rom(sta := BOOL_TO_USINT(REAL_TO_BOOL(xDev^.al.OU.val)) );             // stav
			END_IF;

			// vynuluje koli press, ked Qr sem uz nejde
//			xDev^.al.in.par   := 0;
			cmd					:= 0;

      END_IF;
		nd		:= nd 	+ 1;
   END_WHILE;
END_FUNCTION

FUNCTION _Nh_DEV_RESTART_1  {HIDDEN} :  BOOL   											// kontroly DEV po restarte
	_Nh_DEV_RESTART_1 := true;
	WHILE _Dev_DEV() DO
		IF xDev^.ok.OK THEN
			RETURN;
		END_IF;
	END_WHILE;
	_Nh_DEV_RESTART_1 := false;
END_FUNCTION

VAR_GLOBAL
   rrr   : UDINT;
END_VAR

FUNCTION   _Nh_DEV_RESTART  {HIDDEN} :  BOOL   											// kontroly DEV po restarte
//	aMeteo.WindDelayRol.rst := true;										// resetnut silny vietor

	{$IFDEF __NH_DALI}
  	_Nh_DEV_RESTART := _NH_DEV_INI(c:=44);                            // cf,nd=0,xDev na nd:=0
	WHILE _Nh_DEV_RESTART_1() DO
		xDlg  	:= xDev;
      yTx1  :=  xDev^.cf.Name;
//      REPLACE_CHAR(c1:=16#01,c2:=16#00,input:=yTx1);
      REPLACE_CHAR(c1:=16#01,c2:=16#2C,input:=yTx1);
      REPLACE_CHAR(c1:=16#2C,c2:=16#00,input:=yTx1);
      rrr:=rrr+sz;
      xDev^.cf.Name:=yTx1;
	END_WHILE;
   {$END_IF}

(*
  	_Nh_DEV_RESTART := _NH_DEV_INI(c:=1);                            // cf,nd=0,xDev na nd:=0
	WHILE _Nh_DEV_RESTART_1() DO
		xRom  	:= xDev;
		IF xRom^.cx.IniDefault = false THEN
				xRom^.cx.IniDefault := 1;
				IF xRom^.cx.LuxMin_OLD > 0 AND xRom^.cx.LuxPar.LuxMin = 0 THEN
					xRom^.cx.LuxPar.LuxMin := xRom^.cx.LuxMin_OLD;
				END_IF;
				xRom^.cx.LuxPar.LuxYes	:= 1;
				xRom^.cx.LuxPar.RolYes	:= 1;
				xRom^.io[100].FromZon	:= 1;
				xRom^.io[101].FromZon	:= 1;
				xRom^.io[101].FromOut	:= 1;
				xRom^.io[102].FromZon	:= 1;
				xRom^.cx.LuxPar.KoefBli	:= 1.2;
				xRom^.cx.LuxPar.RolMin	:= 50;
		END_IF;
	END_WHILE;
*)

(*
   _Nh_DEV_RESTART := _NH_DEV_INI(c:=3);                            // cf,nd=0,xDev na nd:=0
	WHILE _Nh_DEV_RESTART_1() DO
		xRom  	:= xDev;
		IF xRom^.cx.IniDefault = false THEN
 			xRom  	:= xDev;
				IF xRom^.cx.LuxMin_OLD > 0 AND xRom^.cx.LuxPar.LuxMin = 0 THEN
					xRom^.cx.LuxPar.LuxMin := xRom^.cx.LuxMin_OLD;
				END_IF;
			xRom^.cx.LuxPar.LuxYes	:= 1;
			xRom^.cx.LuxPar.RolYes	:= 0;
			xRom^.io[100].FromZon	:= 0;
			xRom^.io[101].FromZon	:= 0;
			xRom^.io[101].FromOut	:= 0;
			xRom^.io[102].FromZon	:= 0;
			xRom^.cx.LuxPar.KoefBli	:= 1.0;
		END_IF;
	END_WHILE;
*)

(*
	   _Nh_DEV_RESTART := _NH_DEV_INI(c:=6);                            // HET
		WHILE _Nh_DEV_RESTART_1() DO
			xHet := xDev;
//			IF xHet^.cx.reg.IniDefault = FALSE THEN
			IF true THEN
//				xHet^.cx 					:= eHet.cx;

				FOR i := 0 TO 1 DO
					xHet^.cx.reg.reg[i].hys 					:= eHet.cx.reg.reg[i].hys;
            END_FOR;

//         xHet^.cx.reg.reg[0].req[0] :=  5.0;
//         xHet^.cx.reg.reg[0].req[1] := 20.0;
//         xHet^.cx.reg.reg[0].req[2] := 23.0;
//			xHet^.cx.reg.reg[0].req[3] := 25.0;

				xHet^.cx.reg.IniDefault := true;
			END_IF;

		END_WHILE;

	   _Nh_DEV_RESTART := _NH_DEV_INI(c:=47);                            // HEv
		WHILE _Nh_DEV_RESTART_1() DO
			xHet := xDev;
//			IF xHet^.cx.reg.IniDefault = FALSE THEN
			IF true THEN
//				xHet^.cx.reg 					:= eHev.cx.reg;
//				xHet^.cx 					:= eHev.cx;

				FOR i := 0 TO 1 DO
					xHet^.cx.reg.reg[i].hys 					:= eHet.cx.reg.reg[i].hys;
            END_FOR;

				xHet^.cx.reg.IniDefault := true;
			END_IF;
		END_WHILE;
	   _Nh_DEV_RESTART := _NH_DEV_INI(c:=7);                            // KOT
		WHILE _Nh_DEV_RESTART_1() DO
			xTve := xDev;
//			IF xTve^.cx.reg.IniDefault = FALSE THEN
			IF true THEN
//				xTve^.cx 					:= eKot.cx;

				FOR i := 0 TO 1 DO
					xHet^.cx.reg.reg[i].hys 					:= eHet.cx.reg.reg[i].hys;
            END_FOR;

				xTve^.cx.reg.IniDefault := true;

			END_IF;
		END_WHILE;
	   _Nh_DEV_RESTART := _NH_DEV_INI(c:=8);                            // TVE
		WHILE _Nh_DEV_RESTART_1() DO
			xTve := xDev;
//			IF xTve^.cx.reg.IniDefault = FALSE THEN
			IF true THEN
//				xTve^.cx 					:= eTVE.cx;
				FOR i := 0 TO 1 DO
					xHet^.cx.reg.reg[i].hys 					:= eHet.cx.reg.reg[i].hys;
            END_FOR;

				xTve^.cx.reg.IniDefault := true;
			END_IF;
		END_WHILE;
	   _Nh_DEV_RESTART := _NH_DEV_INI(c:=9);                            // CER
		WHILE _Nh_DEV_RESTART_1() DO
			xTve := xDev;
//			IF xTve^.cx.reg.IniDefault = FALSE THEN
			IF true THEN
//				xTve^.cx 					:= eCER.cx;
				FOR i := 0 TO 1 DO
					xHet^.cx.reg.reg[i].hys 					:= eHet.cx.reg.reg[i].hys;
            END_FOR;

				xTve^.cx.reg.IniDefault := true;
			END_IF;
		END_WHILE;
	   _Nh_DEV_RESTART := _NH_DEV_INI(c:=23);                            // VEN,REK
		WHILE _Nh_DEV_RESTART_1() DO
			xTve := xDev;
//			IF xTve^.cx.reg.IniDefault = FALSE THEN
			IF true THEN
//				xTve^.cx 					:= eVEN.cx;
				FOR i := 0 TO 1 DO
					xHet^.cx.reg.reg[i].hys 					:= eHet.cx.reg.reg[i].hys;
            END_FOR;
				xTve^.cx.reg.IniDefault := true;
			END_IF;
		END_WHILE;

*)

(*
   _Nh_DEV_RESTART := _NH_DEV_INI(c:=31);                            // rolety
	WHILE _Nh_DEV_RESTART_1() DO
 		xRol  	:= xDev;
		IF xRol^.cx.IniDefaul = FALSE THEN
			xRol^.cx.IniDefaul := true;
			xRol^.cx.pLam	:= 0;
			xRol^.cx.uLam	:= 0;
			xRol^.cx.pRol 	:= 0;
			xRol^.cx.uRol	:= 0;
			xRol^.cx.yLam	:= 0.0;
			xRol^.cx.yRol	:= 0.0;
			xRol^.cx.CMD	:= 3;
			xRol^.al.in.val:= 0.0;
			xRol^.al.in.val:= 0.0;
			xRol^.al.ou.val:= 0.0;
			xRol^.cx.NextPar				:= 0;
			xRol^.cx.tStart 				:= UINT_TO_DT(0);
			xRol^.cx.DelayStart  		:= 0;

			xRol^.cx.cf.tUp.Mot 			:= 0;
			xRol^.cx.cf.tUp.chg 			:= 5;
			xRol^.cx.cf.tDn.Mot 			:= 0;
			xRol^.cx.cf.tDn.chg 			:= 5;

			xRol^.cx.cf.tPvHwLam	 	:= 5;
			xRol^.cx.cf.tDelayRev 	:= 10;
			xRol^.cx.cf.tDelayEnd 	:= 2;
			xRol^.cx.cf.LamHWpulse 	 	:= 1;
			xRol^.cx.cf.LamAngle			:= 90;
			xRol^.cx.cf.SetDark 			:= 1;
			xRol^.cx.cf.DarkLam 			:= 40;
			xRol^.cx.cf.DarkRol 			:= 50;
			xRol^.cx.cf.DarkRolLvl 		:= 45;
			xRol^.cx.cf.WindGuardOn		 := true;
			xRol^.cx.cf.WindWaitOn		 := 60;		   					// po akom case [min] pokial presiahne vietor hodnotu [s]
			xRol^.cx.cf.WindWaitOFF		 := 60;                      // ak prestane vietor, po kolkych minutach sa zatiahne tak ako bolo [min]
			xRol^.cx.cf.WindSpeedOn		 := 9;								//	rychlost, pri ktorej sa aktivuje ochrana
			xRol^.cx.cf.WindSpeedOFF	 := 5;								//	rychlost, pri ktorej sa aktivuje koniec ochrany
			xRol^.cx.cf.WindDirFrom	 	 := 0;
			xRol^.cx.cf.WindDirTo	 	 := 360;
			xRol^.cx.cf.WindGuardOn		 := 1;
			xRol^.cx.cf.WindDirOnly		 := 0;
			xRol^.cx.cf.WindGuardBlkTime:= 120;
			xRol^.cx.cf.IgnoreReqLam	:= 5;
			xRol^.cx.cf.IgnoreReqRol	:= 5;

			IF _NhxPar(cp := aCfg[31].par , np := xRol^.cf.par,x:=-1018) THEN
				pRol := xPar;
//				pRol^.SetPozi 	:= false;
				pRol^.all.tDelay 	:= 0;
			END_IF;
		END_IF
	END_WHILE;
  *)

	IF xHom^.cx.IniDefault = false THEN
		xHom^.cx.IniDefault := 1;
	   _Nh_DEV_RESTART := _NH_DEV_INI(c:=1);                            // cf,nd=0,xDev na nd:=0
		WHILE _Nh_DEV_RESTART_1() DO
 			xRom  	:= xDev;
			xRom^.cx.LuxPar.LuxYes	:= 1;
			xRom^.cx.LuxPar.RolYes	:= 1;
			xRom^.io[100].FromZon	:= 1;
			xRom^.io[101].FromZon	:= 1;
			xRom^.io[101].FromOut	:= 1;
			xRom^.io[102].FromZon	:= 1;
			xRom^.cx.LuxPar.LuxMin	:= xRom^.cx.LuxMin_OLD;
			xRom^.cx.LuxPar.RolMin	:= 50;
			xRom^.cx.LuxPar.KoefBli	:= 1.2;
		END_WHILE;
	   _Nh_DEV_RESTART := _NH_DEV_INI(c:=3);                            // cf,nd=0,xDev na nd:=0
		WHILE _Nh_DEV_RESTART_1() DO
 			xRom  	:= xDev;
			xRom^.cx.LuxPar.LuxYes	:= 1;
			xRom^.cx.LuxPar.RolYes	:= 0;
			xRom^.io[100].FromZon	:= 0;
			xRom^.io[101].FromZon	:= 0;
			xRom^.io[101].FromOut	:= 0;
			xRom^.io[102].FromZon	:= 0;
			xRom^.cx.LuxPar.LuxMin	:= xRom^.cx.LuxMin_OLD;
			xRom^.cx.LuxPar.KoefBli	:= 1.0;
		END_WHILE;
	END_IF;

   _Nh_DEV_RESTART := _NH_DEV_INI(c:=40);                            // cf,nd=0,xDev na nd:=0
	WHILE _Nh_DEV_RESTART_1() DO
 		xTgl  	:= xDev;
      xTgl^.cx.cfC.nBTNs 		:= SINT_TO_USINT(xTgl^.cf.typ);
		IF aCfg[cf].ver = 0 THEN
			xTgl^.cx := eTgl.cx;
		END_IF;
   	IF xTgl^.cf.typ = 0 OR xTgl^.cf.typ > 8 THEN
   		xTgl^.cf.typ 	:= 6;
     	END_IF;
		xTgl^.cx.cfL.BtnBli  := LIMIT(xTgl^.cx.cfL.BtnBli,1,SINT_TO_USINT(xTgl^.cf.typ));
		IF xTgl^.cx.cfL.BtnRgb > 3 THEN
	      xTgl^.cx.cfL.BtnRgb 		:= 3;
		END_IF;
(*
      xTgl^.cx.cfL.BtnRgb 		:= 3;
      xTgl^.cx.cfL.dayLvl[0] 	:= 100;
      xTgl^.cx.cfL.dayLvl[1] 	:= 70;
      xTgl^.cx.cfL.dayLvl[2] 	:= 40;
      xTgl^.cx.cfL.dayLvl[3] 	:= 90;
		FOR i := 0 TO 3 DO
	      xTgl^.cx.cfL.DaySlp[i] 	:= 0;
      END_FOR;
      xTgl^.cx.cfL.Sleep 		:= 0;
      xTgl^.cx.cfL.PirRst 		:= 1;
      xTgl^.cx.cfL.PirRst 		:= 1;
*)
      xTgl^.cx.cfL.etSlp	:= -2;
		xTgl^.cx.cfD.etSlp	:= -2;
		xTgl^.cx.cfD.off		:= false;

	END_WHILE;
   _Nh_DEV_RESTART := _NH_DEV_INI(c:=13);                            // cf,nd=0,xDev na nd:=0
	WHILE _Nh_DEV_RESTART_1() DO
 		xTgl  	:= xDev;
		IF aCfg[cf].ver = 0 THEN
			xTgl^.cx := eTgl.cx;
		END_IF;
   	IF xTgl^.cf.typ = 0 OR xTgl^.cf.typ > 8 THEN
   		xTgl^.cf.typ 	:= 2;
     	END_IF;
      xTgl^.cx.cfC.nBTNs 	:= SINT_TO_USINT(xTgl^.cf.typ);
		xTgl^.cx.cfL.BtnBli  := LIMIT(xTgl^.cx.cfL.BtnBli,1,SINT_TO_USINT(xTgl^.cf.typ/2));
      xTgl^.cx.cfL.etSlp	:= -2;
	END_WHILE;

   _Nh_DEV_RESTART := _NH_DEV_INI(c:=14);                            // cf,nd=0,xDev na nd:=0
	WHILE _Nh_DEV_RESTART_1() DO
 		xTGl  	:= xDev;
   	IF xTgl^.cf.typ = 0 OR xTgl^.cf.typ > 5 THEN
   		xTgl^.cf.typ 	:= 1;
     	END_IF;
      xTgl^.cx.cfC.nBTNs 	:= SINT_TO_USINT(xTgl^.cf.typ);
	END_WHILE;

   _Nh_DEV_RESTART := _NH_DEV_INI(c:=6);                            // KOT
	WHILE _Nh_DEV_RESTART_1() DO
 		xDev^.cf.cat := 5;
	END_WHILE;
   _Nh_DEV_RESTART := _NH_DEV_INI(c:=7);                            // KOT
	WHILE _Nh_DEV_RESTART_1() DO
 		xDev^.cf.cat := 39;
	END_WHILE;
   _Nh_DEV_RESTART := _NH_DEV_INI(c:=8);                            // TVE
	WHILE _Nh_DEV_RESTART_1() DO
 		xDev^.cf.cat := 39;
	END_WHILE;
   _Nh_DEV_RESTART := _NH_DEV_INI(c:=9);                            // CER
	WHILE _Nh_DEV_RESTART_1() DO
 		xDev^.cf.cat := 39;
	END_WHILE;

	{$IFDEF __NH_DALI}
(*
   _Nh_DEV_RESTART := _NH_DEV_INI(c:=42);                            // cf,nd=0,xDev na nd:=0
	dlma := 1;
	WHILE _Nh_DEV_RESTART_1() DO
// 		_Nh_DL_ADD_Task(dlm:=dlma, wht := 3, par := 0, sha := 255 ,Block:=true );                       // sta:=  2; pritomnost ballastov
//      _Nh_DL_ADD_Task(dlm:=dlma, wht := 3, par := 1, sha := 255 ,Block:=true );                       // sta:=  3; LVL ballastov
//      _Nh_DL_ADD_Task(dlm:=dlma, wht := 113, par := 16, sha := 255 ,Block:=true );                    //sta:= 4+5  uroven vykonu jedneho SHA v scene: PAR
		dlma := dlma + 1;
	END_WHILE;
*)
   _Nh_DEV_RESTART := _NH_DEV_INI(c:=43);                            // cf,nd=0,xDev na nd:=0
	dlma := 1;
	WHILE _Nh_DEV_RESTART_1() DO
		xDLs	:= xDev;
		xDLs^.me.rmp	:= 99;														// po restarte podhodi nezmyselne cislo
	END_WHILE;
	{$END_IF}
END_FUNCTION

FUNCTION _Nh_TER  {HIDDEN}  : BOOL
   VAR_INPUT
      c     : USINT;
   END_VAR
   _NH_TER := _NH_DEV_INI(c:=c);
   FOR nd := 1 TO aCfg[cf].Rec DO
      IF _Nh_Dev_REC() THEN
     		xTer  := xDev;
			IF xTer^.me.man = false THEN												// VYPNUTE manualne ovladanie cez slider
			   xPtR  := UDINT_TO_PTR(xTer^.hw.d[0]);
//				xDev^.al.IN.val	:= ROUND(xPtR^ * 10.0) / 10.0;   			// zaokruhli na 0.1
				xDev^.al.IN.val	:= xPtR^ ;
			END_IF;
			CASE aSys.RefCyc OF
          	2 : 	// 2.vykonny cyklus - nastavia sa TER,LUX.... aj su ukoncene TypDay pre ZON, Dark od roliet ....
						xDev^.al.vaz := false;			 													// reset priradenia - nastavi sa v ROM/ZON
						xDev^.al.lst := false;			 													// reset priradenia - nastavi sa v ROM/ZON
			END_CASE;

			xTer^.me.f1R (	In 	:= 	xDev^.al.in.val + xTer^.cx.kor ,
								fil	:=    USINT_TO_REAL( xTer^.cx.fil ),	// * 800.0,
								hys	:=		xTer^.cx.hys,
								rst	:= 	xDev^.al.in.cmd = 7 ,	//OR aSys.rst.Qr ,
								sample:=    xTer^.cx.sample,
								Out 	=> 	xDev^.al.OU.val		);										// tu uz pride len s 1.des. miestom

			IF xTer^.me.f1R.Qr OR aSys.RefCyc=2 THEN
//				xDev^.al.OU.val := FLOOR(xTer^.me.f1R.out * 10.0)*0.1;								// pevne 1.des.miesto
				_NhDevRef(xR  := xDev);                                                                        // refresh
				IF xDev^.cf.blk = false THEN
					xDev^.al.OU.cmd   := 100;
					IF xTer^.cx.BlkDefRom = false THEN
						CASE cf OF
							16:	// teplota miestnosti
									xDev^.al.OU.cmd   := 100;
									IF _NhxRom(nr := xDev^.cf.rom ,x:=71) THEN
										_Nh_CHG_VAL(io := ADR( xRom^.io[100] ), val := xDev^.al.ou.val, zon:=false);
						  				_NhDevRef(xR  := xRom);
									END_IF;
	       			END_CASE;
					END_IF;
   			END_IF;
  				_NhDevRef(xR  := xDev);
			END_IF;
		ELSE
			xDev^.al.OU.val := -0.0;
		END_IF;
		xDev^.al.in.cmd 	:= 0;
	END_FOR;
END_FUNCTION

FUNCTION _Nh_LUX  {HIDDEN}  :BOOL
   VAR_INPUT
      c     : USINT;
   END_VAR
   _NH_LUX := _NH_DEV_INI(c:=c);
   FOR nd := 1 TO aCfg[cf].Rec DO
      IF _Nh_Dev_REC() THEN
	   	xLux  := xDev;
         xPtR  := UDINT_TO_PTR(xLux^.hw.d[0]);                                         // default je hodnota v REAL (%)
     	   CASE xLux^.hw.typ OF
         	   2: // INT - LUX,COX...
	               xPtI          	:= xPtR;
   	            vr    			:= INT_TO_REAL(xPtI^);                        //
         	   3: // UINT priamo v luxoch                (C-RI-0401S)
	               xPtUi          := xPtR;
	   	         vr    			:= UINT_TO_REAL(xPtUi^);                        //
         	   4: // USINT 0..255 - uroven osvetlenia    (SOPHY, C-RC-0005R...
            	   xPtU           := xPtR;
	               vr    			:= USINT_TO_REAL(xPtU^);                        //   LUX,COX
   	       ELSE // REAL -45 ... +300
        	      	vr 					:= xPtR^;
     	   END_CASE;
			IF xLux^.me.man = false THEN
	         xLux^.al.in.val := vr;
			END_IF;
			CASE aSys.RefCyc OF
          	2 : 	// 2.vykonny cyklus - nastavia sa TER,LUX.... aj su ukoncene TypDay pre ZON, Dark od roliet ....
						xDev^.al.vaz := false;			 													// reset priradenia - nastavi sa v ROM/ZON
						xDev^.al.lst := false;			 													// reset priradenia - nastavi sa v ROM/ZON
//				3 :	// 3.cyklus po nastaveni typovoveho dna v domceku aj nadradenej zone {zona sa robi pred ROM}
			END_CASE;
			ok := false;
			IF _NhxRom(nr := xDev^.cf.rom ,x:=13) THEN
				// ked sa vypne svetlo, nastartuje sa cakanie na velky reset
				IF cf = 19 AND xRom^.me.Light.Qf THEN							// len pre LUX a po vypnuti svetla v miestnosti
					xLux^.me.nRomQf := xLux^.me.nRomQf + 1;
					xLux^.me.f1R.rstBig	:= true;
				END_IF;
			END_IF;

			xLux^.me.f1R (	In 	:= 	xDev^.al.in.val,
								fil	:=    USINT_TO_REAL( xLux^.cx.fil ),	// * 800.0,
								hys	:=		xLux^.cx.hys,
								sample:=    xLux^.cx.sample,
								rst	:= 	xDev^.al.in.cmd = 7 , //OR aSys.rst.Qr,
								Out 	=> 	xLux^.me.f1R.Out	);

			IF xLux^.me.f1R.Qr OR aSys.RefCyc=2 THEN

IF xLux^.me.f1R.Qr THEN
	xLux^.me.nf1RQr := xLux^.me.nf1RQr + 1;
ELSE
	xLux^.me.nRefCyc := xLux^.me.nRefCyc + 1;
END_IF;

   		      IF xLux^.cx.dark <=  xLux^.cx.sun THEN ;                   		//  dark < sun
      		      vr                := xLux^.cx.Sun 		- xLux^.cx.Dark;     // dark sa presunie na 0... SUN je vacsi  [0....SUN]
         		   kr                := xLux^.me.f1R.Out  - xLux^.cx.Dark;     // upravena filtrovana hodnota
            	 	xLux^.al.ou.val   := kr / Max(vr * 0.01,0.1);      			// % osvetlenia        // spodna hodnota
           		ELSE                                                           // negativny termistor
   		         vr                := (xLux^.cx.Dark 	- xLux^.cx.Sun);     // Sun sa presunie n 0, Sun je mensi      [-SUN.....0]
      		      kr                := (xLux^.me.f1R.Out - xLux^.cx.Sun);
         		   xLux^.al.ou.val   := 100.0 - kr / Max(vr * 0.01,0.1);  		// obratene vyhodnotenie
         	   END_IF;
  	         	xLux^.al.ou.val      := Round(xLux^.al.ou.val);                // % osvetlenia
      	      xLux^.al.ou.val      := LIMIT(0.0,xLux^.al.ou.val,100.0);      // % osvetlenia
					IF xDev^.cf.blk = false THEN      										// nie je BLK posiela sa
						CASE cf OF
                    51: i := 103;	// RH
						  41: i := 102;	// CO2
                  ELSE 	i := 101;	// LUX
                  END_CASE;
						xDev^.al.OU.cmd   := i;
						IF xLux^.cx.BlkDefRom = false THEN									// aj do default ROM
//							IF _NhxRom(nr := xDev^.cf.rom ,x:=13) THEN
								IF xLux^.cx.BlkLuxRom AND xRom^.me.Light.Q THEN
	   							_Nh_CHG_VAL(io := ADR( xRom^.io[i] ), val := xRom^.io[i].val, zon:=false);		// posle existujucu hodnotu, ale zapise, ze ma snimac
								ELSE
	   							_Nh_CHG_VAL(io := ADR( xRom^.io[i] ), val := xDev^.al.ou.val, zon:=false);
					  				_NhDevRef(xR  := xRom);
								END_IF;
//							END_IF;
						END_IF;
   				END_IF;
					xLux^.me.lux		:= xLux^.al.ou.val * xLux^.cx.koef ;
	  				_NhDevRef(xR  := xDev);
			END_IF;
		  	xDev^.al.in.cmd := 0;
		END_IF;
   END_FOR;
END_FUNCTION

FUNCTION _Nh_PIR {HIDDEN} :BOOL
   _NH_PIR := _NH_DEV_INI(c:=15);
   FOR nd := 1 TO aCfg[cf].Rec DO
      IF _NH_DEV_REC() THEN
         xPir              := xDev;                                     // toto len pre filter, ktory pozna len xDev
         IF xDev^.cf.blk = false AND xPir^.hw.d[0] > 0 THEN
            CASE xPir^.cf.typ OF
              1 : // NH analog - signal +70.0, tamper -10.0
                  xPtR  := UDINT_TO_PTR(xPir^.hw.d[0]);
(*
                  ok    := xPtR^ > 70.0; // OR xPtR^ = -40.0;
                  xDev^.al.Off   := xPtR^ > -40.0;                               // zobrazenie bezca pri BLK - ze je elektricky zapojene
                  xDev^.cf.inv   := false;
*)
                  ok    := xPtR^ < -5.0; // OR xPtR^ = -40.0;

              2 : // NH digital - signal pri zopnuti
                  xPtB  := UDINT_TO_PTR(xPir^.hw.d[0]);
                  IF xPir^.cf.inv THEN
                     ok  :=  xPtB^ = false;                                      // signal pri rozopnuti
                  ELSE
                     ok  :=  xPtB^;                                              // signal pri rozopnuti
                  END_IF;

            ELSE  // digital - zopina podla nastavenia
                  xPtB  := UDINT_TO_PTR(xPir^.hw.d[0]);
                  IF xPir^.cf.inv THEN
                     ok  :=  xPtB^ = false;                                      // signal pri rozopnuti
                  ELSE
                     ok  :=  xPtB^;                                              // signal pri rozopnuti
                  END_IF;
            END_CASE;

            IF _Nh_Dev_Qx(In := ok OR xDev^.al.in.cmd = 21 ) THEN       // zabezpeci Qr,Q,Qf, pre prichdzjuce CMD > 0
					_Nh_Log_Evn_ADD( tsk := 15, wht := 'ON ');
               IF xDev^.al.et  > 0 THEN
                  xPir^.al.ou.cmd   := 21;
               ELSIF xPir^.cx.fUnLock = 0 OR xDev^.al.in.cmd = 21 THEN
                  xDev^.al.et       := 1;
                  xDev^.al.Qf       := true;
               ELSE
                  xDev^.al.et       := 100;
                  xDev^.al.ct       := xPir^.cx.funLock*2;
               END_IF;
				ELSIF xDev^.al.trg.Qf THEN
//					_Nh_Log_Evn_ADD( tsk := 15, wht := 'OFF');
            END_IF;
            xDev^.al.in.cmd := 0;
            CASE xDev^.al.et OF
              0 : ;
              1 : IF xDev^.al.Qf OR SYSTEM_S.F_EDGE_1SEC THEN
                     xDev^.al.Qf := false;
                     IF xPir^.al.trg.Q THEN
                        xDev^.al.ou.val   := 100.0;
                        xDev^.al.sta      := 1;
                        xPir^.al.ou.cmd   := 21;
                        xDev^.al.et       := 5;                            // x-SEC po poslednom pohybe bude este zobrazeny pohyb
                     ELSE
                        xDev^.al.et       := 0;
                        xDev^.al.ou.val   := 0.0;
                        xDev^.al.sta      := 0;
                     END_IF;
                     _NhDevRef(xR := xDev);                                 // prvykrat okamzite
                  END_IF;
            100 : // nastartovany filter na pocet cyklov
                  IF xPir^.al.trg.Q THEN
                     IF xDev^.al.ct > xPir^.cx.fUnlock THEN                   // prvykrat nastavi CMD a neskor kazdy 255 cyklus, lebo xPir^.al.ex je USINT co sama resetuje
                        xDev^.al.ct := xDev^.al.ct - 1;
                     ELSE
                        xDev^.al.et       := 1;
                        xDev^.al.Qf       := true;
                     END_IF;
                  ELSE
                     xDev^.al.et       := 0;
                     xDev^.al.ct       := 0;
                  END_IF;
            ELSE
                  xDev^.al.et := xDev^.al.et - aSys.u1Sec;
            END_CASE;
            _Nh_Sta_Rom(sta := REAL_TO_USINT(xDev^.al.ou.val)); //, body :=  );    // stav do miestnosti
         ELSE
            xDev^.al.ou.val := 0.0;
            xDev^.al.sta    := 0;
         END_IF;
      END_IF;
   END_FOR;
END_FUNCTION

(*
                           80,  0,                           //  Ziadna akcia
                          181,  2,                           //  Start/Stop
                          178, 14,                           //  nastavit poziciu
                          180, 25,                           //  Natáèalamely
                          188, 26,                           //  Lamely-potvorit
                          189, 27,                           //  Lamely-Pozatvorit
                          179, 10,                           //  zatiahnut uplne dolu 0%
                          238, 11,                           //  vytiahnut uplne hore 100%
*)

FUNCTION _Nh_DOR  {HIDDEN} :BOOL
   VAR_INPUT
      c    : USINT;
   END_VAR
   cf       := c;
   _Nh_DOR  := _Dev_INI(c := cf);
   FOR nd := 1 TO aCfg[cf].Rec DO
      IF _Nh_Dev_REC(blk:=true) THEN
         xDor  := xDev;
         ok		:= true;
			IF xDev^.cf.DevExt THEN
				;
			ELSIF xDor^.hw.d[0] > 0 THEN
	         xPtB	:= UDINT_TO_PTR(xDor^.hw.d[0]);
			ELSE 	ok	:= false;
			END_IF;
			IF ok THEN
				IF xDev^.cf.inv THEN
					ok	:= xPtB^;
				ELSE
					ok	:= NOT xPtB^;
				END_IF;
	         IF _Nh_Dev_Qx(In := ok OR xDev^.al.in.CMD = 1 ) THEN //  );                                  // zabezpeci Qr,Q,Qf, pre prichdzjuce CMD > 0
					xDev^.al.cm := 2;
					xDev^.al.et := 0;
					_NhxRom(nr:=xDev^.cf.rom);
					IF xDev^.al.in.CMD = 1 THEN
               	;
					ELSIF xRom^.me.Locked THEN
						IF xDor^.cf.psn THEN
							xDev^.al.et := USINT_TO_UINT(xDor^.cx.fLock) * 100;
						END_IF;
					ELSE
						xDev^.al.et := USINT_TO_UINT(xDor^.cx.fUnLock) * 100;		// mSec
					END_IF;
				ELSIF xDev^.al.trg.Qf THEN
					xDev^.al.ou.cmd 	:= 10;  												// off signal
					xDev^.al.cm			:= 0;
					xDev^.al.et 		:= 0;
					_Nh_Sta_Rom(sta := 0);
					_NhDevRef(xR  := xDev);
				END_IF;

				CASE xDev^.al.cm OF
      	      0: // vypnute
						xDev^.al.sta 		:= 0;
						xDev^.al.ou.val   := 0.0;
         	   2: // oneskorenie
						_Nh_Dev_ET(t:=0);														// [mSec]
         	   	IF xDev^.al.et = 0 THEN
							xDev^.al.et 		:= xDor^.cx.tOffRst;
							xDev^.al.cm			:= 100;
         	   	END_IF;
	          100: // zopnute
						_Nh_Dev_ET(t:=1);    												// [sec]
						IF xDev^.al.sta = 0 THEN
	          			xDev^.al.ou.cmd 	:=  14;                          	// on signal
							_Nh_Sta_Rom(sta := 1);
							_NhDevRef(xR  := xDev);
						ELSE
							xDev^.al.sta 		:= 1;
						END_IF;
						xDev^.al.ou.val 	:= 100.0;
      	   ELSE
         	;
	         END_CASE;
   		END_IF;
			IF xDev^.al.ou.cmd > 0 THEN

			END_IF;
			xDev^.al.in.CMD := 0;
      ELSE
         xDev^.al.ou.val   := 0.0;                                      // pir je zablokovany
			xDev^.al.sta 		:= 0;
      END_IF;
	END_FOR;
END_FUNCTION

(*
FUNCTION _Nh_ZON    : BOOL  // ukladanie hodnot do ROM a nasledne do ZON
   _Nh_ZON 				:= _NH_DEV_INI(c:=3);
   xRoW  				:= xHoW;
   FOR nd := 1 TO aCfg[cf].Rec DO
      IF _Nh_Dev_REC() THEN
			xRom								:= xDev;												// aktualna zona
			IF _Nh_Dev_Qx(In := xDev^.al.in.CMD > 0) = false THEN						// LOCK/unLOCK
				IF xRom^.cx.lck.stat	<> xRoW^.LckStat THEN								// zmena stavu alarmu
					IF xRoW^.LckStat = 0 AND xRom^.cx.lck.stat > 1 THEN
						xRom^.al.ou.cmd := 60;           									// prave sa odkodovalo
					ELSIF xRoW^.LckStat = 2 THEN                                   // prave sa zakodovalo
						IF xRom^.cx.lck.stat = 4 THEN
							xRom^.al.ou.cmd := 67;           								// psik zaliezol do budy
						ELSIF xRom^.cx.lck.stat > 4 THEN
							xRom^.al.ou.cmd := 68;           								// obnovenie strazenia zo ALARMU, alebo psik steka
						ELSE
							xRom^.al.ou.cmd := 62;           								// zamknute po odchode
						END_IF;
					ELSE
						xRom^.al.ou.cmd := 60 + xRoW^.LckStat;
					END_IF;
				ELSIF xHoW^.psn AND  xRom^.cx.lck.stat > 3 THEN
					xRom^.al.ou.cmd := 69;													// impulz pri pohybe
				END_IF;

			END_IF;
			xRom^.cx.lck.ChangeStat	:= xRom^.al.ou.cmd > 0;
			IF nd = 1 THEN
				IF xDev^.al.trg.Qr THEN														// domcek sa ma zamknut/odomknut
					IF xRom^.cx.lck.LockRom AND xRom^.cx.lck.stat = 0 THEN      // ak sa zamyka a je odomknute
						xDev^.al.ou.CMD := 56;     										// LOCK
					ELSE
						xDev^.al.ou.CMD := 57;     										// pre istotou unLOCK
					END_IF ;
				END_IF;
         ELSIF _NhxZon(nz := xRom^.cf.rom) THEN                        		// xZon = vyssia domovska zona vyssia zona / Home
				IF xHom^.al.ou.CMD > 0 THEN                                    // v tomto cykle prisiel pokyn z domceka/HOMEzony
					xZon	:= xHom;
					IF xRom^.cx.lck.LockRom THEN											// zona sa centralne zamyka
						xRom^.al.ou.CMD := xZon^.al.ou.CMD;                		// preberie prikaz z HOME
						IF xDev^.al.ou.CMD = 56 THEN						  		   		// len ked Home dava centralne LOCK
							IF xHom^.cx.lck.FromZone THEN								// HOME prepisuje ZON
								xRom^.cx.lck.tdOu	:= xZon^.cx.lck.tdOu;
								xRom^.cx.lck.tdIn	:= xZon^.cx.lck.tdIn;
								xRom^.cx.lck.tDog	:= xZon^.cx.lck.tDog;
								xRom^.cx.lck.tNar	:= xZon^.cx.lck.tNar;
								xRom^.cx.lck.tRst	:= xZon^.cx.lck.tRst;
							END_IF;
						END_IF;
					ELSE
						xDev^.al.ou.CMD := 57;                              		// zona sa centralne nezamyka, pre istotu sa da UNLOCK
					END_IF;

				ELSIF xDev^.al.trg.Qr THEN
					IF xRom^.cx.lck.LockRom AND xRom^.cx.lck.stat = 0 THEN      // ak sa zamyka a je odomknute
						xDev^.al.ou.CMD := 56;     										// LOCK
					ELSE
						xDev^.al.ou.CMD := 57;
					END_IF ;
				END_IF;
			END_IF;
			xRom^.al.in.CMD 				:= 0;
			xRom^.cx.lck.stat				:= xRoW^.LckStat;
			xRom^.cx.lck.et				:= xRoW^.LckEt;
			xRom^.al.sta					:= xRoW^.LckStat;

			xRom^.cx.lck.AllLocked		:= true;              								// nastavi priznak, ze vsetky ROM su locked, neskor sa upravi
			xRom^.me.BodyQr    			:= xRom^.me.BodyQ = false AND xRoW^.body;    // impulz pri zaznamenani pritomnosti
			xRom^.me.BodyQ     			:= xRoW^.body;                         		// pritomnost
			xRom^.me.PsnQr    			:= xRom^.me.PsnQ = false AND xRoW^.psn;      // impulz pri zaznamenani pritomnosti z cidiel PSN
			xRom^.me.PsnQ     			:= xRoW^.psn;// AND xRoW^.LckStat > 1;          // pohyb v zamknutej zone

			CASE aSys.RefCyc OF
				0 :	;
          	2 : 	_Nh_Typ_Day_Fix(xDay:=ADR(xRom^.cx.pDay), go:=xRom^.cf.typ < 2, home:=1);		// 1.vykonny cyklus - len pre domcek alebo byt
				3 :	_Nh_Typ_Day_Fix(xDay:=ADR(xRom^.cx.pDay), go:=xRom^.cf.typ > 1);             // 2.vykonny cyklus - pre ostatne zony
         END_CASE;

//			xRom^.al.lst					:= false;        			            	// resetne priznak zeleneho SETUP zony = ma nejake ROM

			_Nh_IO_VAL(i1:=100, i2:=103, io := ADR(xRom^.io[100]));

          xRom^.al.ou.val := xRom^.io[100].val;

		END_IF;
      xRoW     := xRoW + SIZEOF(NH_WRK_ROM);
   END_FOR;

//	xHom^.me.OldStat	:= xHom^.cx.lck.Stat;

//	xHom^.al.ou.CMD := 0;

END_FUNCTION
*)
(*
FUNCTION _Nh_ZON    : BOOL  // ukladanie hodnot do ROM a nasledne do ZON
   _Nh_ZON 				:= _NH_DEV_INI(c:=3);
   xRoW  				:= xHoW;
   FOR nd := 1 TO aCfg[cf].Rec DO
      IF _Nh_Dev_REC() THEN
			xRom								:= xDev;												// aktualna zona
			IF _Nh_Dev_Qx(In := xDev^.al.in.CMD > 0) = false THEN						// LOCK/unLOCK
				IF xRom^.cx.lck.stat	<> xRoW^.LckStat THEN								// zmena stavu alarmu
					IF xRoW^.LckStat = 0 AND xRom^.cx.lck.stat > 1 THEN
						xRom^.al.ou.cmd := 60;           									// prave sa odkodovalo
					ELSIF xRoW^.LckStat = 2 THEN                                   // prave sa zakodovalo
						IF xRom^.cx.lck.stat = 4 THEN
							xRom^.al.ou.cmd := 67;           								// psik zaliezol do budy
						ELSIF xRom^.cx.lck.stat > 4 THEN
							xRom^.al.ou.cmd := 68;           								// obnovenie strazenia zo ALARMU, alebo psik steka
						ELSE
							xRom^.al.ou.cmd := 62;           								// zamknute po odchode
						END_IF;
					ELSE
						xRom^.al.ou.cmd := 60 + xRoW^.LckStat;
					END_IF;
				ELSIF xHoW^.psn AND  xRom^.cx.lck.stat > 3 THEN
					xRom^.al.ou.cmd := 69;													// impulz pri pohybe
				END_IF;

			END_IF;
			xRom^.cx.lck.ChangeStat	:= xRom^.al.ou.cmd > 0;
			IF nd = 1 THEN
				IF xDev^.al.trg.Qr THEN														// domcek sa ma zamknut/odomknut
					IF xRom^.cx.lck.LockRom AND xRom^.cx.lck.stat = 0 THEN      // ak sa zamyka a je odomknute
						xDev^.al.ou.CMD := 56;     										// LOCK
					ELSE
						xDev^.al.ou.CMD := 57;     										// pre istotou unLOCK
					END_IF ;
				END_IF;
         ELSIF _NhxZon(nz := xRom^.cf.rom) THEN                        		// xZon = vyssia domovska zona vyssia zona / Home
				IF xHom^.al.ou.CMD > 0 THEN                                    // v tomto cykle prisiel pokyn z domceka/HOMEzony
					xZon	:= xHom;
					IF xRom^.cx.lck.LockRom THEN											// zona sa centralne zamyka
						xRom^.al.ou.CMD := xZon^.al.ou.CMD;                		// preberie prikaz z HOME
						IF xDev^.al.ou.CMD = 56 THEN						  		   		// len ked Home dava centralne LOCK
							IF xHom^.cx.lck.FromZone THEN								// HOME prepisuje ZON
								xRom^.cx.lck.tdOu	:= xZon^.cx.lck.tdOu;
								xRom^.cx.lck.tdIn	:= xZon^.cx.lck.tdIn;
								xRom^.cx.lck.tDog	:= xZon^.cx.lck.tDog;
								xRom^.cx.lck.tNar	:= xZon^.cx.lck.tNar;
								xRom^.cx.lck.tRst	:= xZon^.cx.lck.tRst;
							END_IF;
						END_IF;
					ELSE
						xDev^.al.ou.CMD := 57;                              		// zona sa centralne nezamyka, pre istotu sa da UNLOCK
					END_IF;

				ELSIF xDev^.al.trg.Qr THEN
					IF xRom^.cx.lck.LockRom AND xRom^.cx.lck.stat = 0 THEN      // ak sa zamyka a je odomknute
						xDev^.al.ou.CMD := 56;     										// LOCK
					ELSE
						xDev^.al.ou.CMD := 57;
					END_IF ;
				END_IF;
			END_IF;
			xRom^.al.in.CMD 				:= 0;
			xRom^.cx.lck.stat				:= xRoW^.LckStat;
			xRom^.cx.lck.et				:= xRoW^.LckEt;
			xRom^.al.sta					:= xRoW^.LckStat;

			xRom^.cx.lck.AllLocked		:= true;              								// nastavi priznak, ze vsetky ROM su locked, neskor sa upravi
			xRom^.me.BodyQr    			:= xRom^.me.BodyQ = false AND xRoW^.body;    // impulz pri zaznamenani pritomnosti
			xRom^.me.BodyQ     			:= xRoW^.body;                         		// pritomnost
			xRom^.me.PsnQr    			:= xRom^.me.PsnQ = false AND xRoW^.psn;      // impulz pri zaznamenani pritomnosti z cidiel PSN
			xRom^.me.PsnQ     			:= xRoW^.psn;// AND xRoW^.LckStat > 1;          // pohyb v zamknutej zone

			CASE aSys.RefCyc OF
				0 :	;
          	2 : 	_Nh_Typ_Day_Fix(xDay:=ADR(xRom^.cx.pDay), go:=xRom^.cf.typ < 2, home:=1);		// 1.vykonny cyklus - len pre domcek alebo byt
				3 :	_Nh_Typ_Day_Fix(xDay:=ADR(xRom^.cx.pDay), go:=xRom^.cf.typ > 1);             // 2.vykonny cyklus - pre ostatne zony
         END_CASE;

//			xRom^.al.lst					:= false;        			            	// resetne priznak zeleneho SETUP zony = ma nejake ROM

			_Nh_IO_VAL(i1:=100, i2:=103, io := ADR(xRom^.io[100]));

          xRom^.al.ou.val := xRom^.io[100].val;

		END_IF;
      xRoW     := xRoW + SIZEOF(NH_WRK_ROM);
   END_FOR;

//	xHom^.me.OldStat	:= xHom^.cx.lck.Stat;

//	xHom^.al.ou.CMD := 0;

END_FUNCTION
*)

FUNCTION _Nh_ZON   {HIDDEN}   : BOOL  // ukladanie hodnot do ROM a nasledne do ZON
	cf		:= 3;
	xRom	:= xHom;
	xRoW	:= xHoW;
	// najskor sa musia prejst HOME a BYT, lebo BYT	moze byt az za zonou do ktorej patri
   FOR nd := 1 TO aCfg[cf].Rec DO
		IF xRom^.ok.ok AND xRom^.cf.blk = false THEN
			xRom^.me.BodyQr    			:= xRom^.me.BodyQ = false AND xRoW^.body;    // impulz pri zaznamenani pritomnosti
			xRom^.me.BodyQ     			:= xRoW^.body;                         		// pritomnost
			xRom^.me.PsnQr    			:= xRom^.me.PsnQ = false AND xRoW^.psn;      // impulz pri zaznamenani pritomnosti z cidiel PSN
			xRom^.me.PsnQ     			:= xRoW^.psn;// AND xRoW^.LckStat > 1;          // pohyb v zamknutej zone

			IF _Nh_ROM_CMD_IN() THEN
				;
			ELSIF xHom^.al.trg.Qr THEN
				xRom^.al.ou.CMD := xHom^.al.ou.CMD;                   // CMD do zona prebrate z HOM/BYT, kde sa zamyka, aebo bol dotyk
				_Nh_ROM_LOCK_START();
        	ELSIF xRom^.cx.lck.StatOld <> xRom^.cx.lck.Stat THEN
					CASE xRom^.cx.lck.Stat OF
                 	0: // Unlocked
							IF xRom^.cx.lck.StatOld > 1 AND xRom^.cx.lck.AllLockedOld THEN   // len ked sa odomkli vsetky miestnosti naraz
   							xRom^.al.ou.cmd := 60;
                     END_IF;
						1: // odchod - Locking
							xRom^.al.ou.cmd := 61;
                 	2: // Locked
							IF xRom^.cx.lck.StatOld < 2 THEN
	                     xRom^.al.ou.cmd := 62;
							END_IF;
					   3: // prichodove oneskorenie
							xRom^.al.ou.cmd := 63;
					   4: // Dog - ostrazitost
							xRom^.al.ou.cmd := 64;
					   5: // NARUSENIE = tichy poplach
							xRom^.al.ou.cmd := 65;
					   6: // ALARM
							xRom^.al.ou.cmd := 66;
               ELSE
               END_CASE;
				  xRom^.cx.lck.StatOld	:= xRom^.cx.lck.Stat;

         // ak sa miestnosti/zony uzamykanu s inym casom, signal zamknutia sa vysle az ked je zamknuta posledna miestnost
        	ELSIF xRom^.cx.lck.Stat = 2  AND xRom^.cx.lck.AllLocked AND xRom^.cx.lck.AllLockedOld = false THEN
             xRom^.al.ou.cmd := 62;

(*
				CASE xZon^.al.ou.cmd OF
              60: // odomknutie
              61: // zacina zamykanie / zakodovanie;
              62: // zamknute po odchode
              63: // niekto prisiel
              64: // psik z budy von
              65: // psik steka
              66: // ALARM
              67: // Psik zaliezol do budy
              68: // Strazenie obnovene
              69: // pohyb
				ELSE  ok := false;
            END_CASE;
*)

			END_IF;								// bol dotyk nad ZON, moze byt len nad jednou

			xRom^.cx.lck.ChangeStat	   := xRom^.al.ou.cmd > 0;
			xRom^.cx.lck.et 				:= 0;
			xRom^.cx.lck.stat 			:= 0;
			xRom^.cx.lck.AllLockedOld  := xRom^.cx.lck.AllLocked;                   // koli akcie pri LOCK/unLock nie vsetkych miestnosti
			xRom^.cx.lck.AllLocked 		:= true;

			IF xHoW^.chg THEN
				_Nh_ROM_IO_VAL(i1:=100, i2:=103, io := ADR(xRom^.io[100]));
	          xRom^.al.ou.val := xRom^.io[100].val;
				IF nd = 2 THEN																		// vonkajsi sumrak
					aSys.LuxOut := REAL_TO_USINT(xRom^.io[101].val);
				END_IF;
   		END_IF;
			CASE aSys.RefCyc OF
				0 :	;
          	1 : 	_Nh_Typ_Day_Fix(xDay:=ADR(xRom^.cx.pDay), xFix:=ADR(xRom^.cx.FixDay), go:=xRom^.cf.typ < 2, home:=1);		// 1.vykonny cyklus - len pre domcek alebo byt
						xRom^.cx.IniDefault := 1;
				2 :	_Nh_Typ_Day_Fix(xDay:=ADR(xRom^.cx.pDay), xFix:=ADR(xRom^.cx.FixDay), go:=xRom^.cf.typ > 1);             // 2.vykonny cyklus - pre ostatne zony
						_Nh_ROM_Dark();
						// hned za ZON ide ROM, moze sa nastavovat uz v tomto cykle
         END_CASE;
		END_IF;
		xRoM := xRoM + SIZEOF(NH_ROM);
		xRoW := xRoW + SIZEOF(NH_WRK_ROM);
	END_FOR;
END_FUNCTION

FUNCTION _Nh_ROM  {HIDDEN}  :BOOL  // ukladanie hodnot do ROM a nasledne do ZON
	cf			:= 1;
   _NhxRom(nr:=1);																				// xRom
   xRoW  	:= xRoW1;                                                         // xRow
	FOR nd := 1 TO aCfg[cf].Rec DO
		IF xRom^.ok.ok AND xRom^.cf.blk = false THEN
	      xLck 	:= ADR(xRom^.cx.lck);
			_NhxZon(c:=3, nz:=xRom^.cf.Rom, x:=133);											// vyssia zona {xZon, xZow}
(*
			IF xHoW^.chg THEN																		// zmena niektoreho TER/LUX v celom dome
				_Nh_ROM_IO_VAL(clr:=true,i1:=100, i2:=103, io := ADR(xRom^.io[100]));
	          xRom^.al.ou.val := xRom^.io[100].val;
   		END_IF;
*)
			// stav osvetlenia
			_Nh_Qx(in:=xRoW^.cat[1], trg:=ADR(xRom^.me.Light));

			// pritomnost ROM
			xRom^.me.BodyQr    			:= xRom^.me.BodyQ = false AND xRoW^.body;    // impulz pri zaznamenani pritomnosti
			xRom^.me.BodyQ     			:= xRoW^.body;                         		// pritomnost
			xRom^.me.PsnQr    			:= xRom^.me.PsnQ = false AND xRoW^.psn;      // impulz pri zaznamenani pritomnosti z cidiel PSN
			xRom^.me.PsnQ     			:= xRoW^.psn;// AND xRoW^.LckStat > 1;          // pohyb v zamknutej rom
			// rozdelit pritomnost do OUt/In
			IF xRom^.me.BodyQ THEN
				IF xRom^.cf.rom > 2 THEN
					xRoW^.bodyIn 	:= true;
					xZoW^.bodyIn	:= true;
					xHoW^.bodyIn	:= true;
				ELSE
					xRoW^.bodyOu 	:= true;
					xZoW^.bodyOu 	:= true;
					xHoW^.bodyOu 	:= true;
				END_IF;
			END_IF;

			IF xZon^.al.trg.Qr THEN
				xRom^.al.ou.CMD := xZon^.al.ou.CMD;                   // CMD do zona prebrate z HOM/BYT, kde sa zamyka, aebo bol dotyk
				_Nh_ROM_LOCK_START();											// aktualizovat lck.stat
			ELSIF _Nh_ROM_CMD_IN() THEN
					;
			END_IF;

			_Nh_ROM_LOCK_RUN();

			CASE aSys.RefCyc OF
				0 :	;
			  	1 : 	// 1.vykonny cyklus {vacsinou po prechode na novu minutu, alebo rucne v programe}, vynuluju sa lokalne teploty,lux///
						xRom^.cx.IniDefault := 1;
						xRom^.me.DarkRolLvl := 0; 															// resetne sumrak ktory  vdalsom cykle pozbiera z roliet
//	   		       xRom^.al.ou.val := xRom^.io[100].val;
						_Nh_ROM_IO_VAL(clr:=true, i1:=100, i2:=103, io := ADR(xRom^.io[100]));
           	2 : 	// 2.vykonny cyklus - nastavia sa TER,LUX.... aj su ukoncene TypDay pre ZON,
						// nastavil sa aj  xRom^.cx.DarkRolLvl zo vsetkych roliet
						IF NOT(xM^.pod.po.edit.c = cf AND xM^.pod.po.edit.n = nd) THEN
							xRom^.cx.pDay.Day	:= xZon^.cx.pDay.Day;										// natvrdo preberie z vyssej zony
						END_IF;
				3 :	// 3.cyklus po nastaveni typovoveho dna v domceku aj nadradenej zone {zona sa robi pred ROM}
						_Nh_ROM_IO_VAL(i1:=100, i2:=103, io := ADR(xRom^.io[100]));
   		       	xRom^.al.ou.val := xRom^.io[100].val;                                  // teplota miestnosti
//						ELSE
//		   		       xRom^.al.ou.val := -0.0;                                  // teplota miestnosti
//						END_IF;
//            		xPod              := ADR(xRom^.cx.pDay);                          		// namapuje pre dalsie funkcie
		            xRom^.me.DayObr   := INT_TO_SINT(_Nh_Poi_Obr(wh := 0, nd := xRom^.cx.pDay.poi[ xRom^.cx.pDay.day ] )  );
						_Nh_ROM_Dark();
         END_CASE;

         // odpocitava blokovanie vsetkych PIR v miestnsti [min] po vypnuti WSB
			IF _Nh_Dev_ET_USINT(t := 2, et := ADR(xRom^.me.BlPirOff) ) THEN
            _NhDevRef(xR  := xRom);
         END_IF;
			// ak sa nesvieti, blokovanie PIR po zapnuti sa resetne
         IF xRoW^.cat[1] = false  AND xRom^.me.BlPirOn > 0 THEN
				xRom^.me.BlPirOn := xRom^.me.BlPirOn - 1;
			END_IF;
			xRom^.me.Locked := xRom^.cx.lck.stat > 1 ;
			_NhDevRef(xR:=xRom, ref:= xRom^.me.BodyQ <> xRoW^.body OR aSys.RefCyc = 3);
		END_IF;
		xRoM := xRoM + SIZEOF(NH_ROM);
		xRoW := xRoW + SIZEOF(NH_WRK_ROM);
   END_FOR;
END_FUNCTION

(*
FUNCTION _Nh_ROM  :BOOL  // ukladanie hodnot do ROM a nasledne do ZON
   _Nh_ROM 	:= _NH_DEV_INI(c:=1);
   xRoW  	:= xRoW1;
   FOR nd := 1 TO aCfg[cf].Rec DO
      IF _Nh_Dev_REC() THEN
//		  	_Nh_Dev_Qx(In := xRoW^.body);												// Qr = zaciatok pohybu
			xRom					:= xDev;
	      xLck  				:= ADR(xRom^.cx.lck);
			xZon^.al.lst		:= true;

			xRom^.me.BodyQr    			:= xRom^.me.BodyQ = false AND xRoW^.body;    // impulz pri zaznamenani pritomnosti
			xRom^.me.BodyQ     			:= xRoW^.body;                         		// pritomnost
			xRom^.me.PsnQr    			:= xRom^.me.PsnQ = false AND xRoW^.psn;      // impulz pri zaznamenani pritomnosti z cidiel PSN
			xRom^.me.PsnQ     			:= xRoW^.psn;// AND xRoW^.LckStat > 1;          // pohyb v zamknutej rom

         IF _NhxZon(nz := xRom^.cf.rom) THEN                          			// xZon, xZoW
//				xZon^.al.lst := true;
			END_IF;

			IF xRom^.me.BodyQ THEN
				IF xRom^.cf.rom > 2 THEN
					xRoW^.bodyIn 	:= true;
					xZoW^.bodyIn	:= true;
					xHoW^.bodyIn	:= true;
				ELSE
					xRoW^.bodyOu 	:= true;
					xZoW^.bodyOu 	:= true;
					xHoW^.bodyOu 	:= true;
				END_IF;
			END_IF;

			_Nh_IO_VAL(i1:=100, i2:=103, io := ADR(xRom^.io[100]));

	      xRom^.al.ou.val   		:= xRom^.io[100].val;           			// teplota sa prebera v kazdom cykle
			IF xRom^.io[100].chg THEN
		      xRom^.al.ou.CMD   := 100;           			// teplota sa prebera v kazdom cykle
				xRom^.io[100].chg	:= false;
			END_IF;

			_Nh_ROM_LOCK();

			CASE aSys.RefCyc OF
				0 :	;
				1 :   // nastartuje refresh
			  	2 : 	// 1.vykonny cyklus {vacsinou po prechode na novu minutu, alebo rucne v programe}, vynuluju sa lokalne teploty,lux///
          	3 : 	// 2.vykonny cyklus - nastavia sa TER,LUX....
				4 :	// 4.cyklus po nastaveni typovoveho dna v domceku aj nadradenej zone

            		xPod              := ADR(xRom^.cx.pDay);                          	// namapuje pre dalsie funkcie
						IF xM^.pod.po.edit	= false THEN
							xPod^.Day			:= xZon^.cx.pDay.Day;									// natvrdo preberie z vyssej zony
						END_IF;
		            xRom^.me.DayObr   := INT_TO_SINT(_Nh_Poi_Obr(wh := 0, nd := xPod^.poi[ xPod^.day] )  );

		            IF xRom^.cx.LuxMin = 0 THEN                               					// sumrak sa moze zadat rucne
      	            xRom^.cx.Dark := true;
         		   ELSIF xRom^.io[101].val < USINT_TO_REAL(xRom^.cx.LuxMin) THEN          // osvetlenei je < ako nastavene minimum = je sumrak
               	   xRom^.cx.Dark := true;
		            ELSIF xRom^.io[101].val >= USINT_TO_REAL(xRom^.cx.LuxMin) THEN         // je svetlo
      	            xRom^.cx.Dark := false;
   	      	   END_IF;
						xRom^.cx.Dark 		:= xRom^.cx.Dark OR xRom^.cx.DarkBli;						// akceptuje aj rolety
						xRom^.me.ClearBli	:= false;															// resetne priznak pre nastavovanie Dark Rolety

				5 :
         END_CASE;

         IF aSys.Cyc_F_Min = 4 THEN													// 3. cyklus po ptrrchode na novu minutu
//				xRom^.cx.pDay.Day  := xZon^.cx.pDay.Day ;
				_Nh_TypDay(xDay:=ADR(xRom^.cx.pDay), xFix:=ADR(xRom^.cx.pDay.Fix), go:=true);

            j                 := xRom^.me.DayObr;                             // len si zapamata stary obrazok, koli zmene
            xPod              := ADR(xRom^.cx.pDay);                          // namapuje pre dalsie funkcie
				xRom^.cx.pDay.day := LIMIT(xRom^.cx.pDay.day,1,11);

            xRom^.me.DayObr   := INT_TO_SINT(_Nh_Poi_Obr(wh := 0, nd := xRom^.cx.pDay.poi[xRom^.cx.pDay.day] )  );
            _NhDevRef(xR:=xRom, ref:= j <> xRom^.me.DayObr);
            // zistenie sumraku
            ok2 := xRom^.cx.Dark;
            IF xRom^.cx.LuxMin = 0 THEN                               					// sumrak sa moze zadat rucne
                  xRom^.cx.Dark := true;
            ELSIF xRom^.io[101].val < USINT_TO_REAL(xRom^.cx.LuxMin) THEN          // osvetlenei je < ako nastavene minimum = je sumrak
                  xRom^.cx.Dark := true;
            ELSIF xRom^.io[101].val >= USINT_TO_REAL(xRom^.cx.LuxMin) THEN         // je svetlo
                  xRom^.cx.Dark := false;
            END_IF;
				xRom^.cx.Dark := xRom^.cx.Dark OR xRom^.cx.DarkBli;					// akceptuje aj rolety
				xRom^.me.ClearBli	:= false;													// resetne priznak pre nastavovanie Dark Rolety
            _NhDevRef(xR  := xRom, ref := ok2 <> xRom^.cx.Dark);
         END_IF;
         // alarm
         // odpocitava blokovanie vsetkych PIR v miestnsti [min] po vypnuti WSB
			IF _Nh_Dev_ET_USINT(t := 2, et := ADR(xRom^.me.BlPirOff) ) THEN
            _NhDevRef(xR  := xRom);
         END_IF;
			// ak sa nesvieti, blokovanie PIR po zapnuti sa resetne
         IF xRoW^.cat[1] = false  AND xRom^.me.BlPirOn > 0 THEN
				xRom^.me.BlPirOn := xRom^.me.BlPirOn - 1;
			END_IF;
      END_IF;
		xRom^.me.Locked := xRom^.cx.lck.stat > 1 ;
		_NhDevRef(xR:=xRom, ref:= xRom^.me.BodyQ <> xRoW^.body OR aSys.RefCyc = 5);
      xRoW  :=  xRoW + SIZEOF(NH_WRK_ROM);
   END_FOR;
END_FUNCTION
*)

FUNCTION _Nh_ACT    : BOOL
   _Nh_ACT := _Dev_INI(c := 5);
   WHILE _Dev_DEV() DO
      IF xDev^.ok.ok THEN
         xDev^.al.lst   	:= 0;
         xDev^.al.ou.cmd   := 0;

         IF _Nh_Dev_Qx(in := xDev^.al.in.cmd > 0) THEN
				xDev^.al.RMP 		:= xDev^.al.in.cmd;											// len pre ladenie co prislo
				IF xDev^.al.in.cmd = 1 THEN
					xDev^.al.in.cmd := 14;
				END_IF;

				xDev^.al.cm 		:= xDev^.al.in.cmd;
				IF xDev^.cf.typ = 1 THEN															//ROLETY
		(*
					CASE xDev^.al.cm OF
	  					10:	// vytiahnut hore
								xDev^.al.Up			:= false;
								xDev^.al.ou.val 	:= BOOL_TO_REAL(xDev^.al.Up); 						// na zaciatku nastavi vsetky rolety rovnakym smerom
								xDev^.al.cm			:= 23;
	  					11:	// zatiahnut dolu
								xDev^.al.Up			:= true;
								xDev^.al.ou.val 	:= BOOL_TO_REAL(xDev^.al.Up); 						// na zaciatku nastavi vsetky rolety rovnakym smerom
								xDev^.al.cm			:= 23;
	  					14:	// predvolena pozicia
								;
	  					23:	// z SCN - centralne START/STOP
								xDev^.al.Up		:= NOT xDev^.al.Up;
								xDev^.al.ou.val := BOOL_TO_REAL(xDev^.al.Up); 						// na zaciatku nastavi vsetky rolety rovnakym smerom
					  	24:	// z SCN -  centralne naklapat lameny
								xDev^.al.Up		:= NOT xDev^.al.Up;
								xDev^.al.ou.val := BOOL_TO_REAL(xDev^.al.Up); 						// na zaciatku nastavi vsetky rolety rovnakym smerom
					END_CASE;
*)
				END_IF;

				xDev^.al.ou.cmd 	:= xDev^.al.cm;			//xDev^.al.in.cmd;                                      // vypina sa
            xDev^.al.sta 	 	:= 1;
            xDev^.al.et 	 	:= 10;														// 30  x 100ms = 3s
				xDev^.al.wsb 		:= false;																// akcia nie je WSB, vykona sa okamzite

				IF xDev^.al.in.cmd = 1 THEN												// ked sa akcia spusti z WEB, tiez moze blokovat PIR
//					xDev^.al.wsb := true;
//					xDev^.al.wsb := false;													// web neblokuje
				ELSE
               ;
				END_IF;
            _NhDevRef(xR  := xDev);
				If xDev^.cf.LogAct THEN
					_Nh_Log_Evn_ADD(tsk:=-1, evn:='ACT', wht:='BEG', val1:=USINT_TO_STRINGF(xDev^.al.IN.cmd,'%7u'), val2:=USINT_TO_STRINGF(xDev^.al.OU.cmd,'%7u'));
   			END_IF;
			ELSIF xDev^.al.trg.Q  THEN
				IF xDev^.al.cm = 24 OR xDev^.al.cm = 6 THEN							// stmievat,natacat rolety
					xDev^.al.ou.cmd := xDev^.al.cm;
				ELSE
					xDev^.al.wsb := false;
   			END_IF;
			ELSIF xDev^.al.trg.Qf  THEN
				xDev^.al.wsb 		:= false;
            xDev^.al.ou.val 	:= 0.0;                                       // pre istotu sa nuluje, aj ked by nemalo mat vplyv, lebo vDEV sa nastavi LVL z parametra

			ELSIF _Nh_Dev_ET(t := 3) AND xDev^.al.Qf  THEN
         	_NhDevRef(xR  := xDev);
            xDev^.al.sta 	 := 0;
         END_IF;
//         xDev^.al.in.val := xDev^.al.ou.val;
         xDev^.al.in.cmd := 0;
      END_IF;
   END_WHILE;
END_FUNCTION

FUNCTION _NH_HET   {HIDDEN}   : BOOL
   VAR_INPUT
      c  : USINT;
   END_VAR
   _NH_HET := _NH_DEV_INI(c:=c);

   FOR nd := 1 TO aCfg[cf].Rec DO
//   FOR nd := 1 TO MIN(1,aCfg[cf].Rec) DO
		IF _NH_Het_CMD() THEN
				// TVE
				xPtIO 	:= ADR(xHet^.io[1]);									         // TVE
				IF _Nh_IO_DEV(io := xPtIO, val := false) THEN	       			// mapuje TVE, ale neodcita teplotu, lebo ta nie je v xDev^.al.ou.Val, ale xTve^.io[1].val
					xTve := xPt;
					_Nh_CHG_VAL(io := xPtIO, val := xTve^.io[1].val, zon := xTve^.io[1].own);   // do zon sa zapise, ci ma TVE teplotu
					xTve^.al.in.par	:= MAX(xTve^.al.in.par, USINT_TO_INT(xHet^.me.Out));
					IF xTve^.cx.reg.ModeFromSrc THEN
						xTve^.cx.reg.Mode 		 := xHet^.cx.reg.Mode;
					END_IF;
				END_IF;
				// KOT
				xPtIO 	:= ADR(xHet^.io[2]);									         			// KOT
				IF _Nh_IO_DEV(io := xPtIO, val := false) THEN
					xTve := xPt;
					_Nh_CHG_VAL(io := xPtIO, val := xTve^.io[1].val, zon := xTve^.io[1].own);
					xTve^.al.in.par	:= MAX(xTve^.al.in.par, USINT_TO_INT(xHet^.me.Out));   // do zon sa zapise, ci ma KOT teplotu
					IF xHet^.cx.reg.ModeFromSrc THEN
						xHet^.cx.reg.Mode			 := xTve^.cx.reg.Mode;
					END_IF;
				END_IF;
				// CER
				xPtIO 	:= ADR(xHet^.io[3]);									         			// CER
				IF _Nh_IO_DEV(io := xPtIO, val := false) THEN
					xTve := xPt;
					_Nh_CHG_VAL(io := xPtIO, val := xTve^.io[1].val);
					xTve^.al.in.par	:= MAX(xTve^.al.in.par, USINT_TO_INT(xHet^.me.Out));
					IF xTve^.cx.reg.ModeFromSrc THEN
						xTve^.cx.reg.Mode 		 := xHet^.cx.reg.Mode;
					END_IF;
				END_IF;

//			xHet^.cf.cat := 39;													// setup kurenia, do het zapisuju ventily

			_Nh_Sta_Rom(sta := xHet^.al.sta) ;             				// stav do

			_NH_Het_LOG();

		ELSE
			xHet^.al.sta 			:= 0;
		END_IF;
   END_FOR;
END_FUNCTION

FUNCTION _NH_TVE    {HIDDEN}   :BOOL
   VAR_INPUT
      c  : USINT;
   END_VAR
   _NH_TVE := _NH_DEV_INI(c:=c);
   FOR nd := 1 TO aCfg[cf].Rec DO
//   FOR nd := 1 TO MIN( 1,aCfg[cf].Rec ) DO
		IF _NH_TVE_CMD() THEN
(*
			IF xTve^.cx.PWM THEN                         								// riadenie PWM ma prednost
			END_IF;
*)
			CASE xTve^.me.CMD OF
   			0:	// pokoj, alebo pohyb
					IF xTve^.cf.typ = 1 AND cf = 8 THEN													/// TECO
						xTvTecoIn 			:= UDINT_TO_PTR(xTve^.hw.d[0]);
						xTvTecoOu 			:= UDINT_TO_PTR(xTve^.hw.d[1]);
						xTve^.me.stat		:= xTvTecoIn^;										// prenesie status TV do mem
						IF xDev^.al.IN.val <> xTvTecoOu^.POSITION THEN           	// niekto iny zmenil HW alebo ext.App
							xDev^.al.in.val	:= xTvTecoOu^.POSITION;						// preberie sa hodnota aby sa v dalsom cykle zapis

							xPvA^.p.pv 			:= _NH_TVE_VAL_TO_PV();               	// vypocita sa priblizne PV

							xPvA^.p.prg			:= false;                              //
						ELSIF xTvTecoIn^.POSITION <> xTvTecoOu^.POSITION THEN
							_NhDevRef(xR := xDev);
						END_IF;
						xDev^.al.OU.val	:= xTvTecoIn^.POSITION;
					ELSIF xDev^.al.OU.val = xDev^.al.IN.val THEN
						;
					ELSIF xTve^.cx.guard.tRun > 0 THEN                                 	// ostatne TVE
						_NhInkrValTst(wh:=1, cj:=2, tRun:=xTve^.cx.guard.tRun, in:=ADR(xTve^.al.in.Val), ou:=ADR(xTve^.al.ou.Val) );
						_NhDevRef(xR := xDev);
					 ELSE
  						xTve^.al.ou.val 		:= xTve^.al.in.val;
						_NhDevRef(xR := xDev);
					END_IF;
				1: // nema HW adresu
					;

           10: // nastavenie
					xTve^.me.CMD := 0;														// default je ze sa pojde zatvarat
					IF xTve^.cf.typ = 1 AND cf = 8 THEN                         // len TVE TECO
						IF xTve^.hw.d[1]	> 0 THEN
							xTvTecoOu 				:= UDINT_TO_PTR(xTve^.hw.d[1]);
							xTvTecoOu^.POSITION	:= xDev^.al.IN.val;
						ELSE
							xTve^.me.CMD := 1;
						END_IF;
					ELSIF xTve^.io[0].dev.c = 43 THEN										// DALI TVE
						_NhxPt(c:=xTve^.io[0].dev.c, n:=xTve^.io[0].dev.n);		// xDLs
						xDls := xPt;
						IF xDev^.al.IN.val > 0.0 THEN
							ii 	:= 254;
						ELSE
							ii		:= 0;
						END_IF;
						i := xTve^.io[0].dev.o;													// 0..5  (0-R-G-B-W-A)
						IF  i > 0 THEN                                              // je zlozka
						   _NhxPar2 (cp := aCfg[ xTve^.io[0].dev.c ].par , np := xPt^.cf.par);	// default parameter xDLs
							xTve^.io[0].val 	:= USINT_TO_REAL(ii);
							IF xPar2^.rgb.lvl[i] <> ii OR xDLs^.me.SendDLM = false THEN// zlozka je ina ako sa pozaduje, alebo ete nebol poslany prikaz

								xDLs^.al.in.cmd	:= 143;
								xDLs^.al.in.par := 0;
								xDLs^.al.in.val := UDINT_TO_REAL( PTR_TO_UDINT(ADR(xTve^.io[0])) );	// posle sa cela struktura
							END_IF;
						ELSE																			// 1 SHA
							xPt^.al.in.cmd		:= 11;
							xPt^.al.in.val		:= MIN(254,xDev^.al.IN.val * 2.54);
							xDLs^.al.in.par 	:= 0;
						END_IF;

					ELSIF xTve^.hw.d[0] > 0 THEN												// fyzicky poslat do HW
		      	   xPtB	:= UDINT_TO_PTR(xTve^.hw.d[0]);
						ok 	:= REAL_TO_BOOL(xDev^.al.IN.val);							// predpripavi na BOOL
						CASE xTve^.hw.typ  OF        											// toto si oznaci sam export
                    0 :  // BOOL
								_Nh_Tve_Obr_OnOff(off	:= true,        					// najskor vypne ine rele. ktore by bolo zapnute
												lvl 	:= xTve^.me.pvm.p.pv,                 // zapne konkretny stupen
												inv	:= xTve^.cf.Inv,                    // zohladni ci su rele inverne
												hw:=ADR(xTve^.hw), reg:=ADR(xTve^.cx.reg));
								// ak hw[1] {PV-1} musi zosta zapnute - pri rekuperacii
								IF xTve^.cx.guard.PV1_IsOn AND xTve^.me.pvm.p.pv > 1 THEN
		      	   			xPtB	:= UDINT_TO_PTR(xTve^.hw.d[0]);
	      	   				xPtB^	:= true;
								END_IF
	                 1 : // REAL
								xPtr	:= xPtB;
								xPtR^ := xDev^.al.IN.val;

                  ELSE	 // ostatne sa bude brat ze maju nespravnu adresu
								xTve^.me.CMD := 1;
                  END_CASE;
					ELSE
						xTve^.me.CMD := 1;														// nema hw adresu
					END_IF;
       	END_CASE;
			IF xDev^.al.ou.val = 0.0 THEN
				xDev^.al.sta := 0;
			ELSE
				_Nh_Sta_Rom(sta := xPvA^.p.pv);    // stav do miestnosti
			END_IF;

      END_IF;
   END_FOR;
END_FUNCTION

(* Ikony  xKy001Ou^.icons
   0  Lock
   1  Unlock
   2  Lock + vykricnik
   4

*)

(*
FUNCTION _Nh_KEY_BEEP  {HIDDEN} : BOOL
   VAR_INPUT
      set   : BOOL;
      end   : BOOL;
      nx    : USINT  := 2;
      et    : UINT   := 500;
   END_VAR
   IF end THEN
      xDev^.al.el    := 0;
      xDev^.al.et    := 1000;
      xDev^.al.CM    := 99;
      xDev^.al.Up    := 0;
      xDev^.al.rmp   := 0;
   ELSIF set THEN
      xDev^.al.el    := xKey^.cx.tMax;
      xDev^.al.et    := et;
      xDev^.al.ct    := 0;
      xDev^.al.Up    := 0;
      xDev^.al.rmp   := nx;
   ELSIF xDev^.al.rmp > 0 THEN
      xDev^.al.rmp   := xDev^.al.rmp - 1;
      xDev^.al.Up    := NOT xDev^.al.Up;
      xDev^.al.et    := et;
   ELSE
      xDev^.al.et    := 1000;
      IF xDev^.al.cm = 2 THEN
         xDev^.al.CM    := 202;
      ELSE
         xDev^.al.CM    := 200;
      END_IF;
      xDev^.al.Up    := 0;
   END_IF;

   IF xDev^.al.Up THEN
      CASE xDev^.cf.typ OF
         1: xKy001Ou^.SETT := USINT_TO_BYTE(3);          // zapne BEEP
      ELSE
            xWg503Ou^.DOs.DO2 := 0;                      // zapne cervenu
            xWg503Ou^.DOs.DO1 := 1;                      // Beep ON
      END_CASE;
   ELSIF xDev^.cf.typ = 1 THEN
      xKy001Ou^.SETT := USINT_TO_BYTE(1);          // vypne BEEP
   ELSE
      xWg503Ou^.DOs.DO2 := 1;                      // zapne zltu
      xWg503Ou^.DOs.DO1 := 0;                      // Beep OFF
   END_IF;
END_FUNCTION
*)

FUNCTION _Nh_KEY_PIN {HIDDEN}  : BOOL
	FOR  i := 1 TO INT_TO_USINT(aCfg[22].rec) DO
 		IF _NhxUsr(u := i) THEN
			ix := LEN(xKey^.me.KeyPas);
	      IF ix >=3 AND xUsr^.cx.keyPas = xKey^.me.KeyPas THEN
				xKey^.me.keyPas 	:= '';
				_Nh_KEY_PIN 		:= true;
				RETURN;
			END_IF;
		END_IF;
   END_FOR;
	_Nh_KEY_PIN := false;
END_FUNCTION

FUNCTION _Nh_KEY {HIDDEN}    : BOOL
   VAR_INPUT
      c  : USINT := 24;
   END_VAR
   _NH_KEY := _NH_DEV_INI(c:=c);
   FOR nd := 1 TO aCfg[cf].Rec DO
      IF _Nh_Dev_REC(blk:=true) THEN
			xDev^.al.Off		:= false;												// naslo sa helso
         xKey  				:= xDev;
         xRom 					:= xHom;
			xLck					:= ADR(xHom^.cx.lck);
			xDev^.al.ou.CMD   := 0;
//			xKey^.me.Qf			:= false;												// pusteny btn
//			xKey^.me.Q			:= false;                                   	// drzime btn
			xKey^.me.ChgTx1	:= 0;
			xKey^.me.ChgTx2	:= 0;
			y						:= LEN(xKey^.me.keyPas);							// pocet zadanych znakov
         xDev^.al.sta 		:= xHom^.cx.lck.stat;
(*
				CASE xZon^.al.ou.cmd OF
              60: // odomknutie
              61: // zacina zamykanie / zakodovanie;
              62: // zamknute po odchode
              63: // niekto prisiel
              64: // psik z budy von
              65: // psik steka
              66: // ALARM
              67: // Psik zaliezol do budy
              68: // Strazenie obnovene
              69: // pohyb
				ELSE  ok := false;
            END_CASE;
*)
			i	:= 0;
			ii := 1;																				// rozvieteny display

			_Nh_Dev_ET();                                                  // odcitava al.et 500 ms filter pre dalsie odcitanie stlacenie

			IF _Nh_Dev_ET_USINT(t:=1, et:=ADR(xDev^.al.cm)) THEN           // odcitava cas zobrazenia hesla
				IF y > 0 OR xDev^.al.sta = 0 THEN
					xKey^.me.keyPas 	:= '';
					yTx1					:= '';
					xKey^.me.ChgTx2 	:= 1;
				END_IF;
			END_IF;
			IF xHom^.me.bodyQ  THEN                                     	// trva pohyb
//				yTx1 := '';
//				_Nh_ALARM_ROM();															// zoznam, kde je pohyb vlozi do yTx1
				xKey^.me.ChgTx2	:= 1;
				IF y = 0 THEN
					xDev^.al.cm	:= 5;			                                 // heslo je prazdne, podhadzuje sa 5s
				END_IF;
			END_IF;
			IF xHom^.cx.lck.ChangeStat OR aSys.Restart THEN						// zmena stavu PSN, restart
				_NhxPt(c:=48, n := USINT_TO_INT(xHom^.cx.lck.stat+1), x:=344 );
				yTx2					:= xPt^.cf.Name;
				xKey^.me.ChgTx1	:= 1;
				IF xHom^.al.ou.cmd = 60  THEN                     				// odomknutie
					xKey^.me.beep.wht := 102;
					xKey^.me.beep.nbr := 2;
					xKey^.me.ChgTx2 	:= 1;
					yTx1					:= '';
				ELSIF xHom^.al.ou.cmd = 62 OR       // zamknutie
						xHom^.al.ou.cmd = 67 OR       // psik zaliezol do budy
						xHom^.al.ou.cmd = 68 THEN    	// obnovenie po alarme
					xKey^.me.beep.wht := 102;
					xKey^.me.beep.nbr := 3;
					xKey^.me.ChgTx2 	:= 1;
					yTx1					:= '';
				ELSIF xHom^.al.ou.cmd = 69 THEN 										// pohyb v zamknutej zone
					xKey^.me.beep.wht := 102;
					xKey^.me.beep.nbr := 3;
  				END_IF;
			ELSIF xDev^.al.sta = 0  THEN
				;
			ELSIF xDev^.al.sta = 1 OR (xDev^.al.sta=2 AND xHom^.cx.lck.et > 0) THEN // zamykam alebo je uz zamknute ale vonkajsie zony sa este zamykaju
				IF aSys.PULSE_BEEP THEN
					ii := 67;	// 1 + 2 + 64;											// podsvietenie aj pipanie
				ELSE
					ii := 65;																// len podsvietenie
				END_IF;
			ELSIF xDev^.al.sta = 3 THEN												// Narusenie
				IF SYSTEM_S.PERIOD_PULSE_1SEC THEN
					ii := 67;	// 1 + 2 + 64;
				ELSE
					ii := 65;	//1 + 0 + 64;
				END_IF;
			END_IF;
			IF xKey^.me.beep.wht <> 0 THEN                 						// beeper ma prednost
				IF xKey^.me.beep.Q THEN
					ii := 67;
				ELSE
					ii := 65;
				END_IF;
			END_IF;
